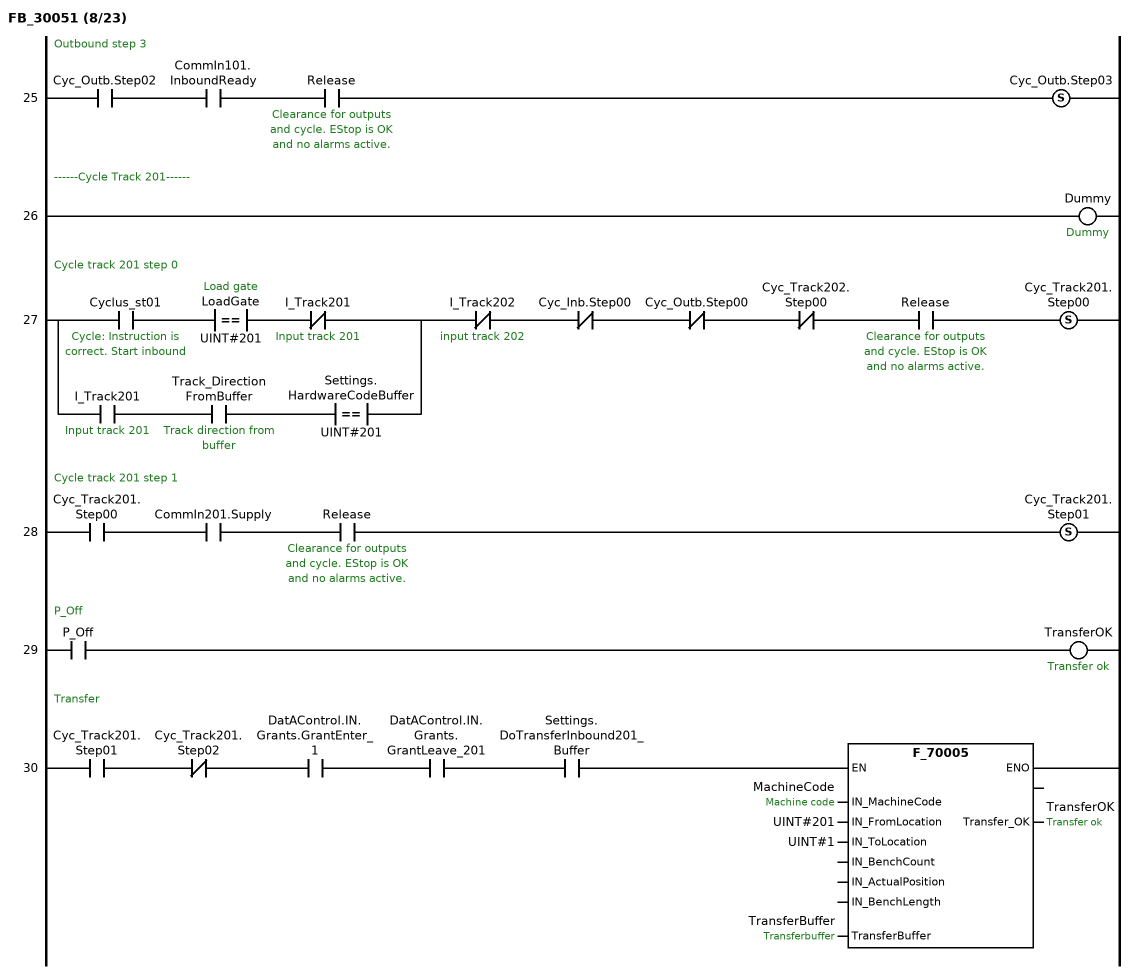
(* Rung 25: Outbound step 3 *)
IF Cyc_Outb.Step02 AND CommIn101.InboundReady AND Release THEN Cyc_Outb.Step03 := TRUE; END_IF;
(* Rung 26: ------Cycle Track 201------ *)
Dummy := TRUE;
(* Rung 27: Cycle track 201 step 0 *)
IF ((Cyclus_st01 AND (LoadGate = UINT#201) AND NOT I_Track201) OR (I_Track201 AND Track_DirectionFromBuffer AND (Settings.HardwareCodeBuffer = UINT#201))) AND NOT I_Track202 AND NOT Cyc_Inb.Step00 AND NOT Cyc_Outb.Step00 AND NOT Cyc_Track202.Step00 AND Release THEN
    Cyc_Track201.Step00 := TRUE;
END_IF;
(* Rung 28: Cycle track 201 step 1 *)
IF Cyc_Track201.Step00 AND CommIn201.Supply AND Release THEN Cyc_Track201.Step01 := TRUE; END_IF;
(* Rung 29: P_Off *)
TransferOK := P_Off;
(* Rung 30: Transfer *)
IF Cyc_Track201.Step01 AND NOT Cyc_Track201.Step02 AND DatAControl.IN.Grants.GrantEnter_1 AND DatAControl.IN.Grants.GrantLeave_201 AND Settings.DoTransferInbound201_Buffer THEN
    F_70005(IN_MachineCode := MachineCode, IN_FromLocation := UINT#201, IN_ToLocation := UINT#1, TransferBuffer := TransferBuffer, Transfer_OK => TransferOK);
END_IF;

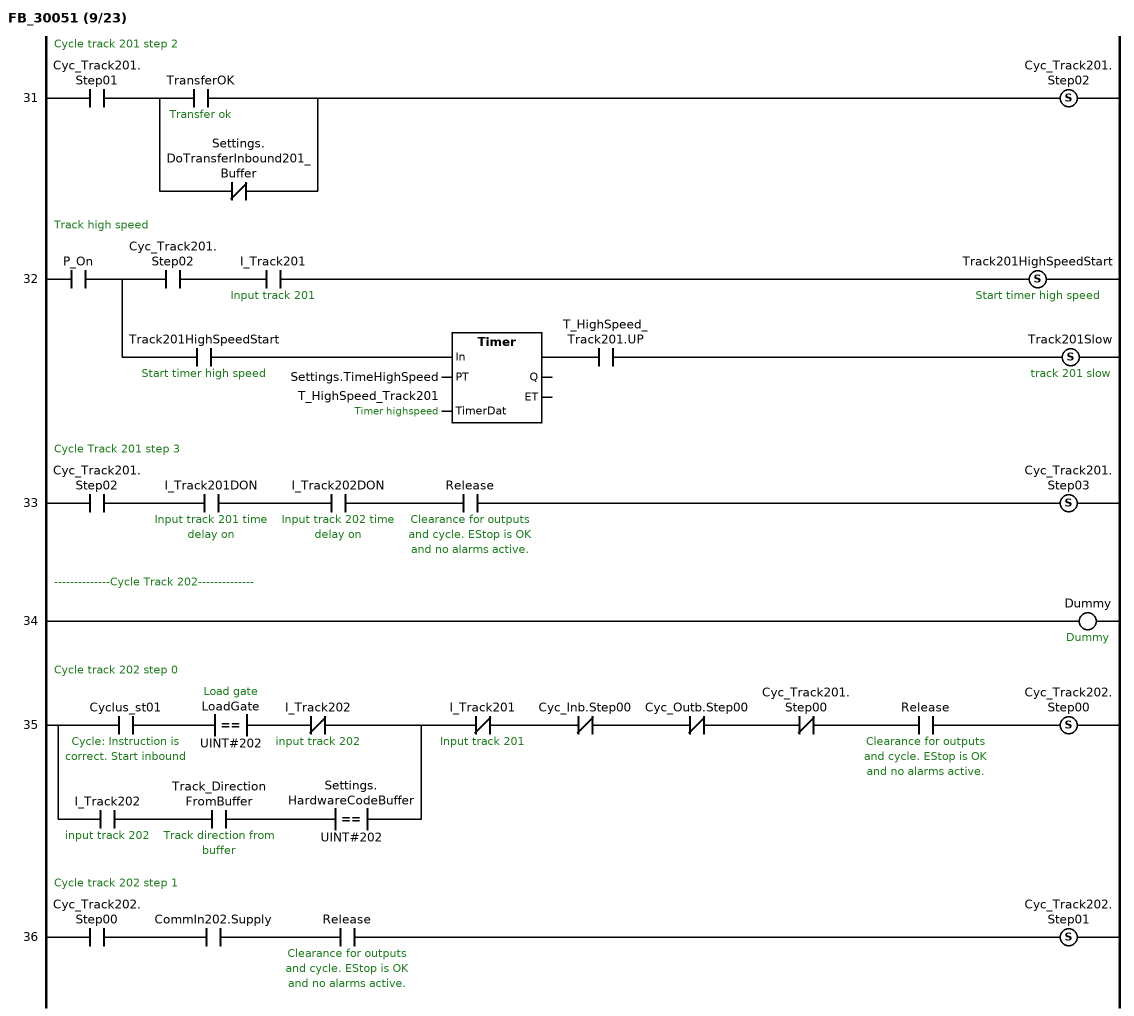
(* Rung 31: Cycle track 201 step 2 *)
IF Cyc_Track201.Step01 AND (TransferOK OR NOT Settings.DoTransferInbound201_Buffer) THEN
    Cyc_Track201.Step02 := TRUE;
END_IF;
(* Rung 32: Track high speed *)
IF P_On AND Cyc_Track201.Step02 AND I_Track201 THEN Track201HighSpeedStart := TRUE; END_IF;
_t2 := Timer(In := P_On AND Track201HighSpeedStart, PT := Settings.TimeHighSpeed, TimerDat := T_HighSpeed_Track201);
IF _t2 AND T_HighSpeed_Track201.UP THEN Track201Slow := TRUE; END_IF;
(* Rung 33: Cycle Track 201 step 3 *)
IF Cyc_Track201.Step02 AND I_Track201DON AND I_Track202DON AND Release THEN
    Cyc_Track201.Step03 := TRUE;
END_IF;
(* Rung 34: --------------Cycle Track 202-------------- *)
Dummy := TRUE;
(* Rung 35: Cycle track 202 step 0 *)
IF ((Cyclus_st01 AND (LoadGate = UINT#202) AND NOT I_Track202) OR (I_Track202 AND Track_DirectionFromBuffer AND (Settings.HardwareCodeBuffer = UINT#202))) AND NOT I_Track201 AND NOT Cyc_Inb.Step00 AND NOT Cyc_Outb.Step00 AND NOT Cyc_Track201.Step00 AND Release THEN
    Cyc_Track202.Step00 := TRUE;
END_IF;
(* Rung 36: Cycle track 202 step 1 *)
IF Cyc_Track202.Step00 AND CommIn202.Supply AND Release THEN Cyc_Track202.Step01 := TRUE; END_IF;

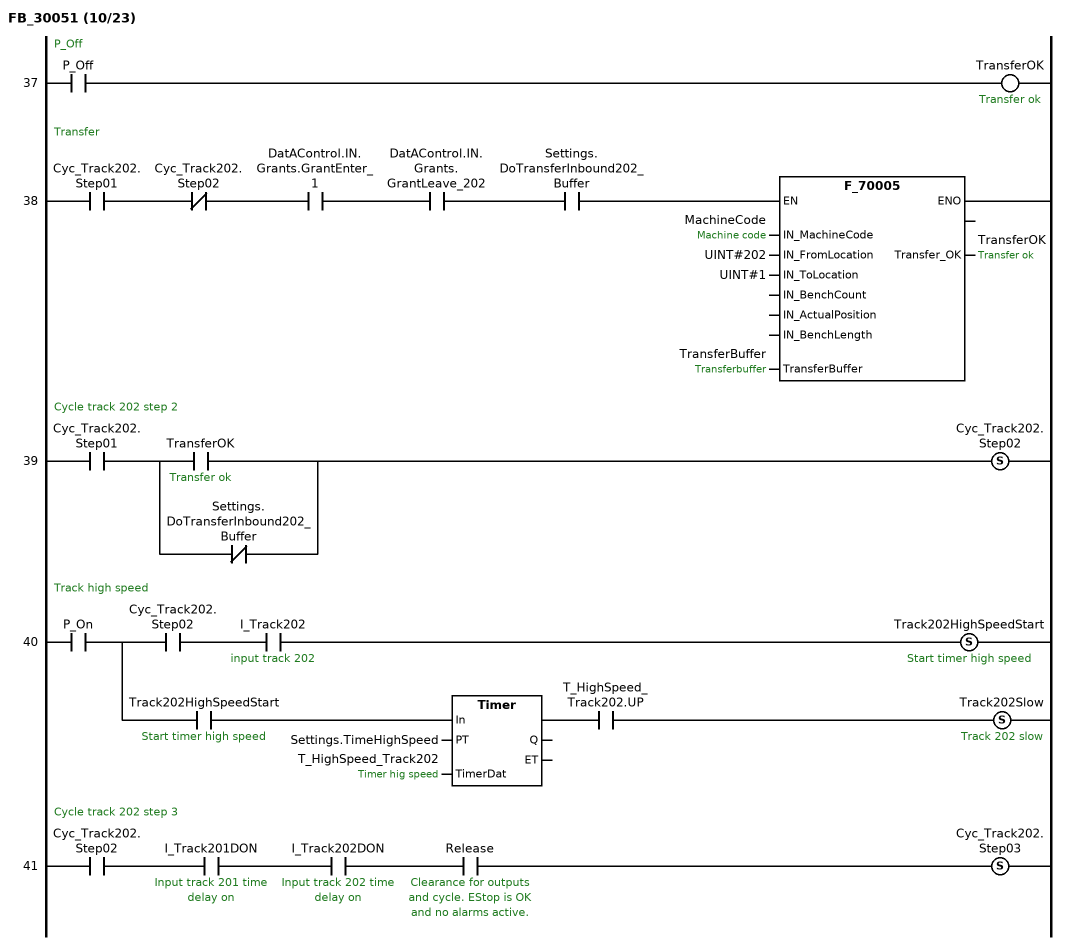
(* Rung 37: P_Off *)
TransferOK := P_Off;
(* Rung 38: Transfer *)
IF Cyc_Track202.Step01 AND NOT Cyc_Track202.Step02 AND DatAControl.IN.Grants.GrantEnter_1 AND DatAControl.IN.Grants.GrantLeave_202 AND Settings.DoTransferInbound202_Buffer THEN
    F_70005(IN_MachineCode := MachineCode, IN_FromLocation := UINT#202, IN_ToLocation := UINT#1, TransferBuffer := TransferBuffer, Transfer_OK => TransferOK);
END_IF;
(* Rung 39: Cycle track 202 step 2 *)
IF Cyc_Track202.Step01 AND (TransferOK OR NOT Settings.DoTransferInbound202_Buffer) THEN
    Cyc_Track202.Step02 := TRUE;
END_IF;
(* Rung 40: Track high speed *)
IF P_On AND Cyc_Track202.Step02 AND I_Track202 THEN Track202HighSpeedStart := TRUE; END_IF;
_t3 := Timer(In := P_On AND Track202HighSpeedStart, PT := Settings.TimeHighSpeed, TimerDat := T_HighSpeed_Track202);
IF _t3 AND T_HighSpeed_Track202.UP THEN Track202Slow := TRUE; END_IF;
(* Rung 41: Cycle track 202 step 3 *)
IF Cyc_Track202.Step02 AND I_Track201DON AND I_Track202DON AND Release THEN
    Cyc_Track202.Step03 := TRUE;
END_IF;

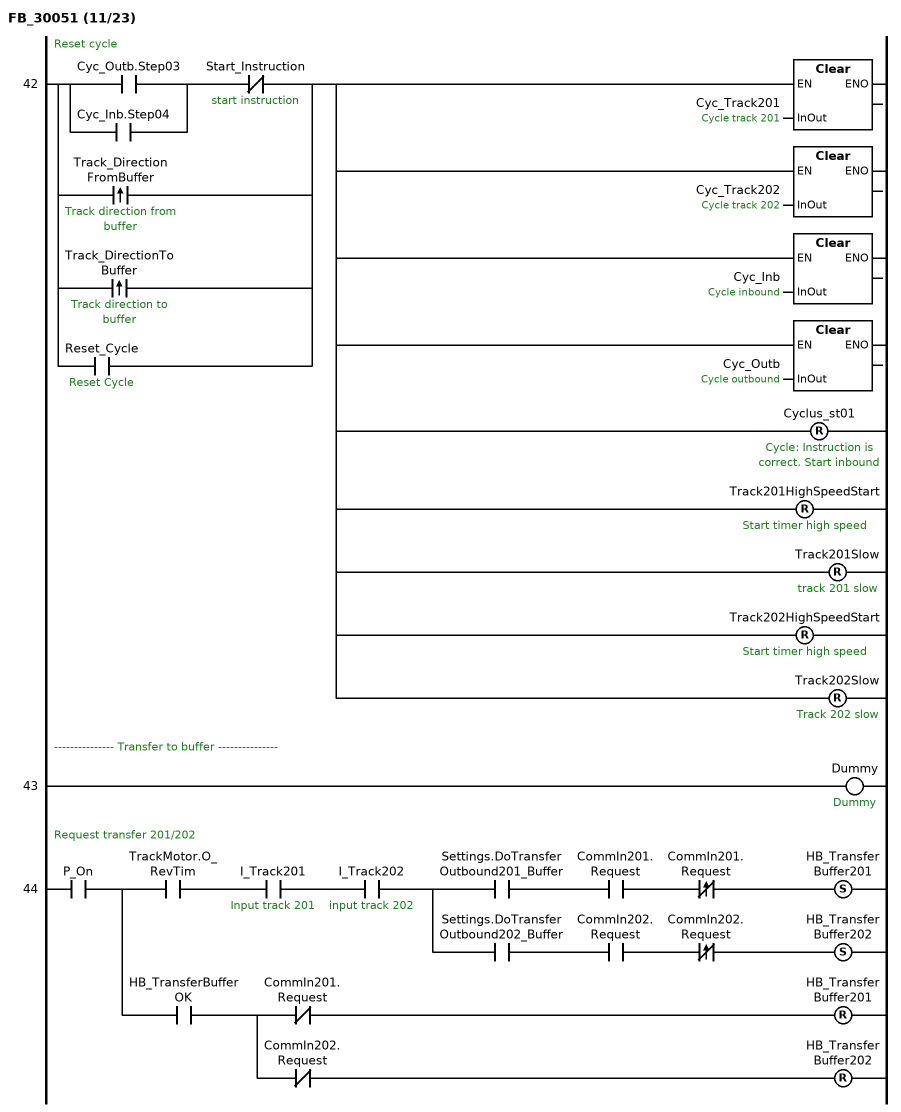
(* Rung 42: Reset cycle *)
_e4(CLK := Track_DirectionFromBuffer);
_e5(CLK := Track_DirectionToBuffer);
_p6 := ((Cyc_Outb.Step03 OR Cyc_Inb.Step04) AND NOT Start_Instruction) OR _e4.Q OR _e5.Q OR Reset_Cycle;
IF _p6 THEN
    Clear(InOut := Cyc_Track201);
    Clear(InOut := Cyc_Track202);
    Clear(InOut := Cyc_Inb);
    Clear(InOut := Cyc_Outb);
    Cyclus_st01 := FALSE;
    Track201HighSpeedStart := FALSE;
    Track201Slow := FALSE;
    Track202HighSpeedStart := FALSE;
    Track202Slow := FALSE;
END_IF;
(* Rung 43: --------------- Transfer to buffer --------------- *)
Dummy := TRUE;
(* Rung 44: Request transfer 201/202 *)
_p7 := P_On AND TrackMotor.O_RevTim AND I_Track201 AND I_Track202;
_e8(CLK := CommIn201.Request);
IF _p7 AND Settings.DoTransferOutbound201_Buffer AND CommIn201.Request AND NOT _e8.Q THEN
    HB_TransferBuffer201 := TRUE;
END_IF;
_e9(CLK := CommIn202.Request);
IF _p7 AND Settings.DoTransferOutbound202_Buffer AND CommIn202.Request AND NOT _e9.Q THEN
    HB_TransferBuffer202 := TRUE;
END_IF;
IF P_On AND HB_TransferBufferOK AND NOT CommIn201.Request THEN HB_TransferBuffer201 := FALSE; END_IF;
IF P_On AND HB_TransferBufferOK AND NOT CommIn202.Request THEN HB_TransferBuffer202 := FALSE; END_IF;

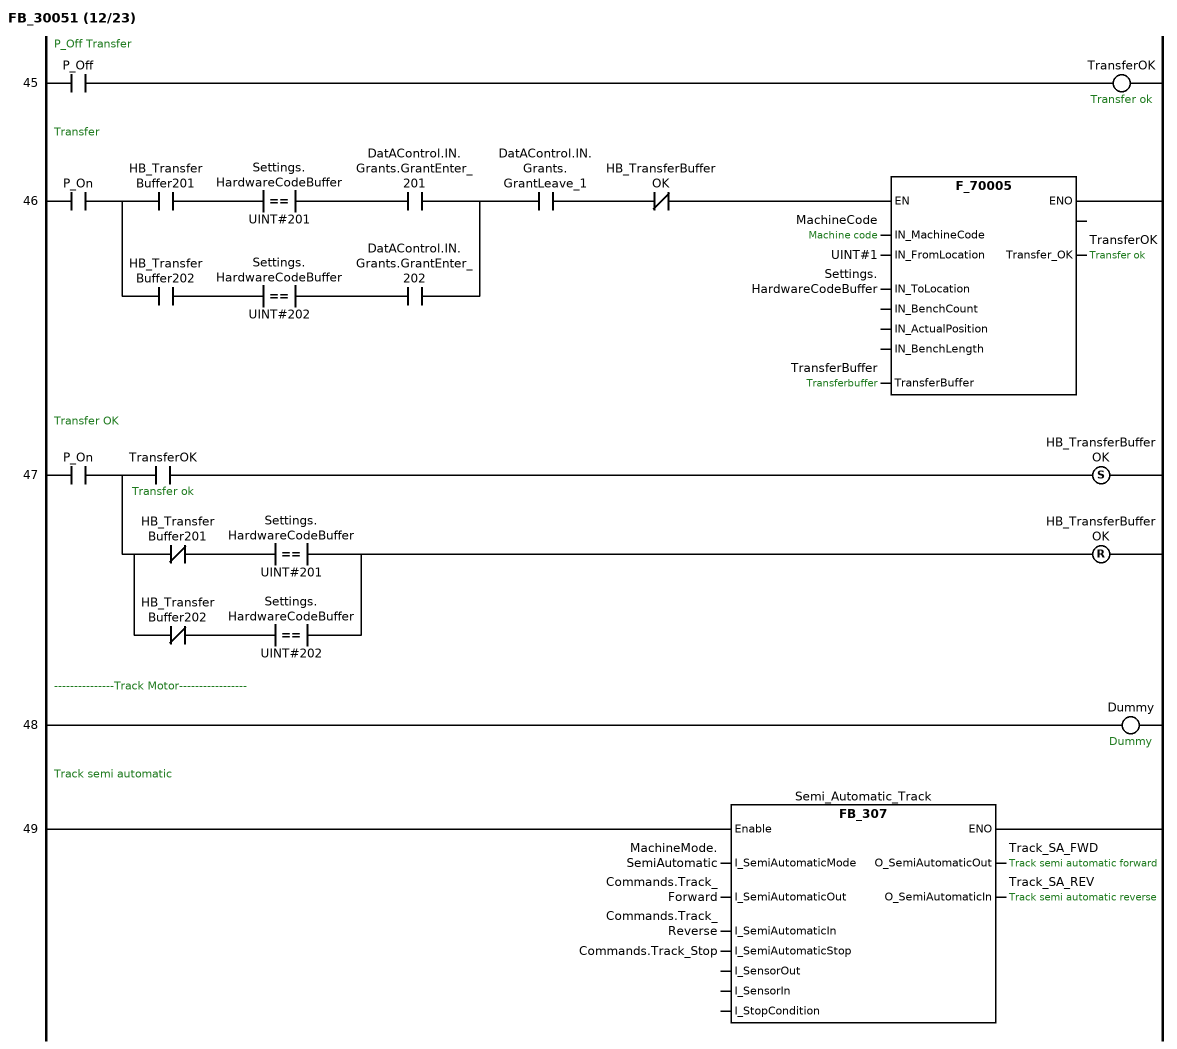
(* Rung 45: P_Off Transfer *)
TransferOK := P_Off;
(* Rung 46: Transfer *)
IF P_On AND ((HB_TransferBuffer201 AND (Settings.HardwareCodeBuffer = UINT#201) AND DatAControl.IN.Grants.GrantEnter_201) OR (HB_TransferBuffer202 AND (Settings.HardwareCodeBuffer = UINT#202) AND DatAControl.IN.Grants.GrantEnter_202)) AND DatAControl.IN.Grants.GrantLeave_1 AND NOT HB_TransferBufferOK THEN
    F_70005(IN_MachineCode := MachineCode, IN_FromLocation := UINT#1, IN_ToLocation := Settings.HardwareCodeBuffer, TransferBuffer := TransferBuffer, Transfer_OK => TransferOK);
END_IF;
(* Rung 47: Transfer OK *)
IF P_On AND TransferOK THEN HB_TransferBufferOK := TRUE; END_IF;
IF P_On AND ((NOT HB_TransferBuffer201 AND (Settings.HardwareCodeBuffer = UINT#201)) OR (NOT HB_TransferBuffer202 AND (Settings.HardwareCodeBuffer = UINT#202))) THEN
    HB_TransferBufferOK := FALSE;
END_IF;
(* Rung 48: ---------------Track Motor----------------- *)
Dummy := TRUE;
(* Rung 49: Track semi automatic *)
Semi_Automatic_Track(Enable := TRUE, I_SemiAutomaticMode := MachineMode.SemiAutomatic, I_SemiAutomaticOut := Commands.Track_Forward, I_SemiAutomaticIn := Commands.Track_Reverse, I_SemiAutomaticStop := Commands.Track_Stop, O_SemiAutomaticOut => Track_SA_FWD, O_SemiAutomaticIn => Track_SA_REV);

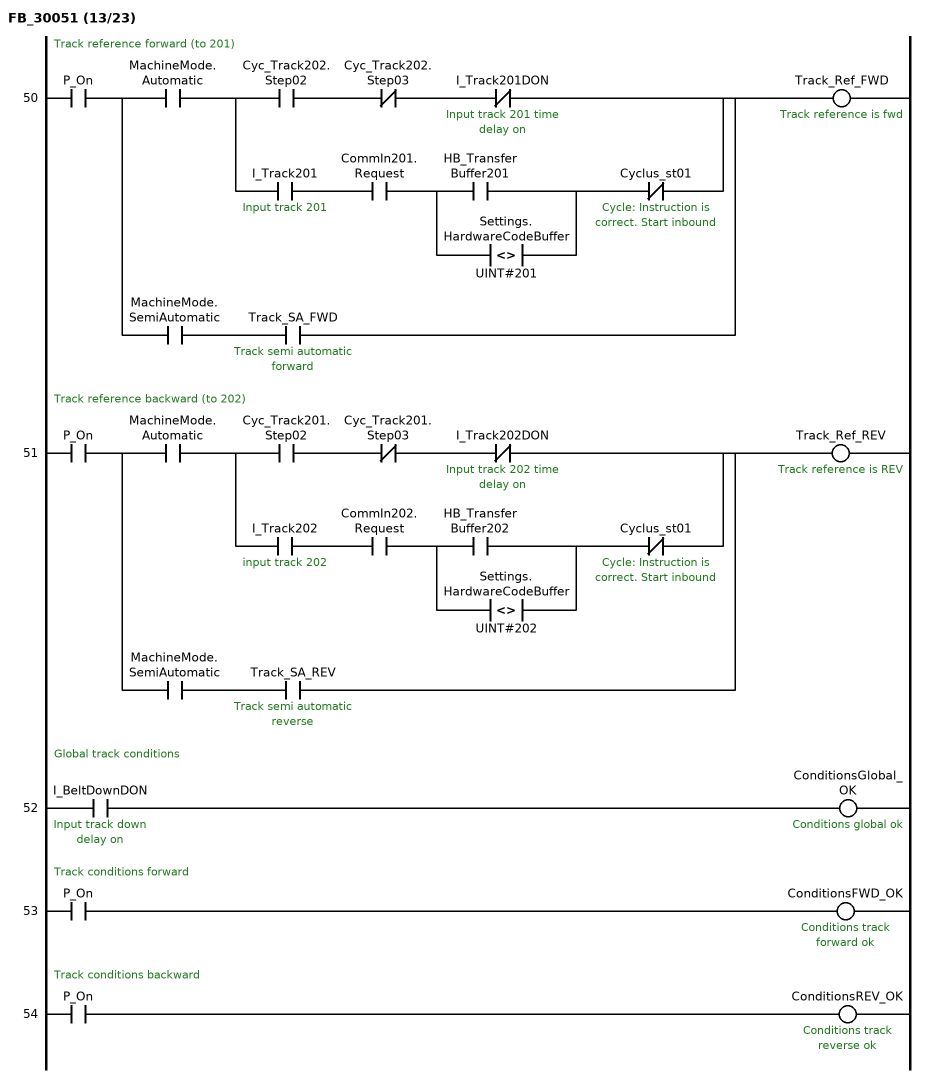
(* Rung 50: Track reference forward (to 201) *)
Track_Ref_FWD := P_On AND ((MachineMode.Automatic AND ((Cyc_Track202.Step02 AND NOT Cyc_Track202.Step03 AND NOT I_Track201DON) OR (I_Track201 AND CommIn201.Request AND (HB_TransferBuffer201 OR (Settings.HardwareCodeBuffer <> UINT#201)) AND NOT Cyclus_st01))) OR (MachineMode.SemiAutomatic AND Track_SA_FWD));
(* Rung 51: Track reference backward (to 202) *)
Track_Ref_REV := P_On AND ((MachineMode.Automatic AND ((Cyc_Track201.Step02 AND NOT Cyc_Track201.Step03 AND NOT I_Track202DON) OR (I_Track202 AND CommIn202.Request AND (HB_TransferBuffer202 OR (Settings.HardwareCodeBuffer <> UINT#202)) AND NOT Cyclus_st01))) OR (MachineMode.SemiAutomatic AND Track_SA_REV));
(* Rung 52: Global track conditions *)
ConditionsGlobal_OK := I_BeltDownDON;
(* Rung 53: Track conditions forward *)
ConditionsFWD_OK := P_On;
(* Rung 54: Track conditions backward *)
ConditionsREV_OK := P_On;

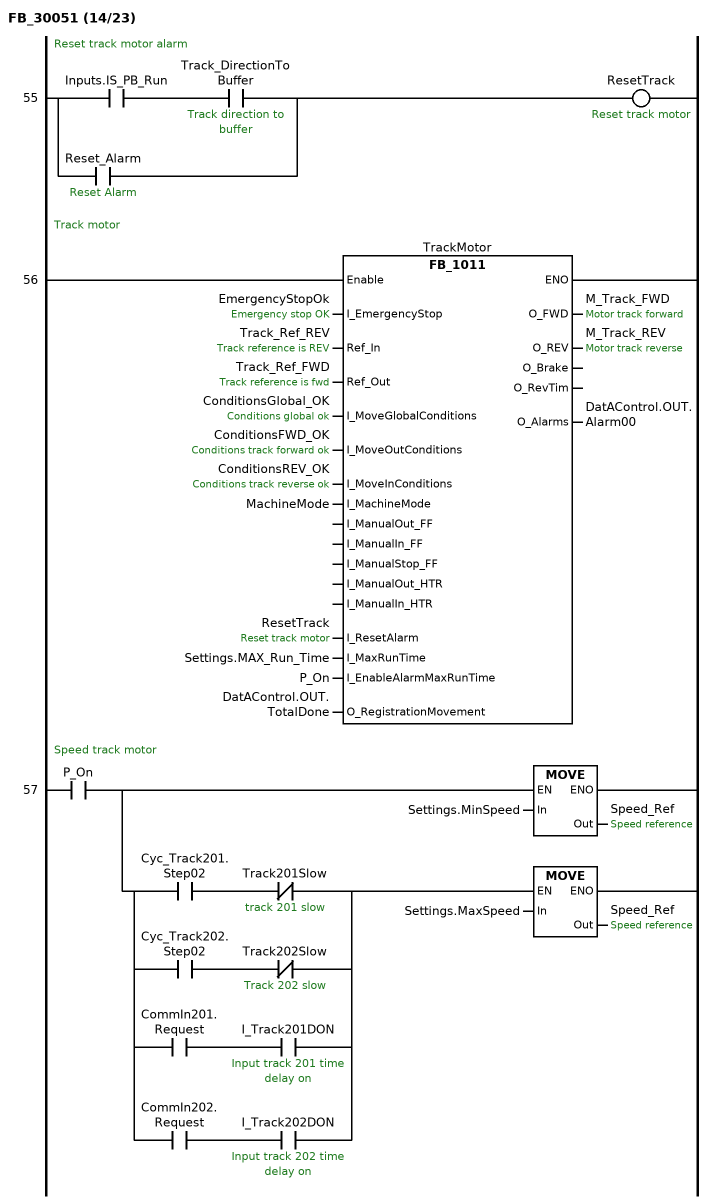
(* Rung 55: Reset track motor alarm *)
ResetTrack := (Inputs.IS_PB_Run AND Track_DirectionToBuffer) OR Reset_Alarm;
(* Rung 56: Track motor *)
TrackMotor(Enable := TRUE, I_EmergencyStop := EmergencyStopOk, Ref_In := Track_Ref_REV, Ref_Out := Track_Ref_FWD, I_MoveGlobalConditions := ConditionsGlobal_OK, I_MoveOutConditions := ConditionsFWD_OK, I_MoveInConditions := ConditionsREV_OK, I_MachineMode := MachineMode, I_ResetAlarm := ResetTrack, I_MaxRunTime := Settings.MAX_Run_Time, I_EnableAlarmMaxRunTime := P_On, O_RegistrationMovement := DatAControl.OUT.TotalDone, O_FWD => M_Track_FWD, O_REV => M_Track_REV, O_Alarms => DatAControl.OUT.Alarm00);
(* Rung 57: Speed track motor *)
IF P_On THEN Speed_Ref := Settings.MinSpeed; END_IF;
IF P_On AND ((Cyc_Track201.Step02 AND NOT Track201Slow) OR (Cyc_Track202.Step02 AND NOT Track202Slow) OR (CommIn201.Request AND I_Track201DON) OR (CommIn202.Request AND I_Track202DON)) THEN
    Speed_Ref := Settings.MaxSpeed;
END_IF;

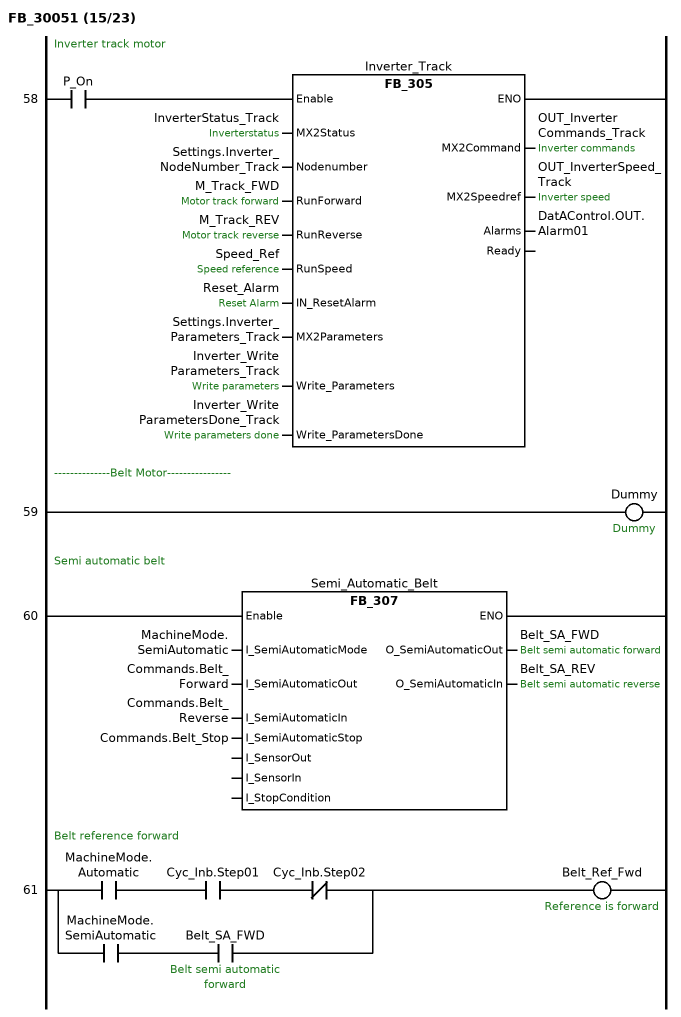
(* Rung 58: Inverter track motor *)
Inverter_Track(Enable := P_On, MX2Status := InverterStatus_Track, Nodenumber := Settings.Inverter_NodeNumber_Track, RunForward := M_Track_FWD, RunReverse := M_Track_REV, RunSpeed := Speed_Ref, IN_ResetAlarm := Reset_Alarm, MX2Parameters := Settings.Inverter_Parameters_Track, Write_Parameters := Inverter_WriteParameters_Track, Write_ParametersDone := Inverter_WriteParametersDone_Track, MX2Command => OUT_InverterCommands_Track, MX2Speedref => OUT_InverterSpeed_Track, Alarms => DatAControl.OUT.Alarm01);
(* Rung 59: --------------Belt Motor---------------- *)
Dummy := TRUE;
(* Rung 60: Semi automatic belt *)
Semi_Automatic_Belt(Enable := TRUE, I_SemiAutomaticMode := MachineMode.SemiAutomatic, I_SemiAutomaticOut := Commands.Belt_Forward, I_SemiAutomaticIn := Commands.Belt_Reverse, I_SemiAutomaticStop := Commands.Belt_Stop, O_SemiAutomaticOut => Belt_SA_FWD, O_SemiAutomaticIn => Belt_SA_REV);
(* Rung 61: Belt reference forward *)
Belt_Ref_Fwd := (MachineMode.Automatic AND Cyc_Inb.Step01 AND NOT Cyc_Inb.Step02) OR (MachineMode.SemiAutomatic AND Belt_SA_FWD);

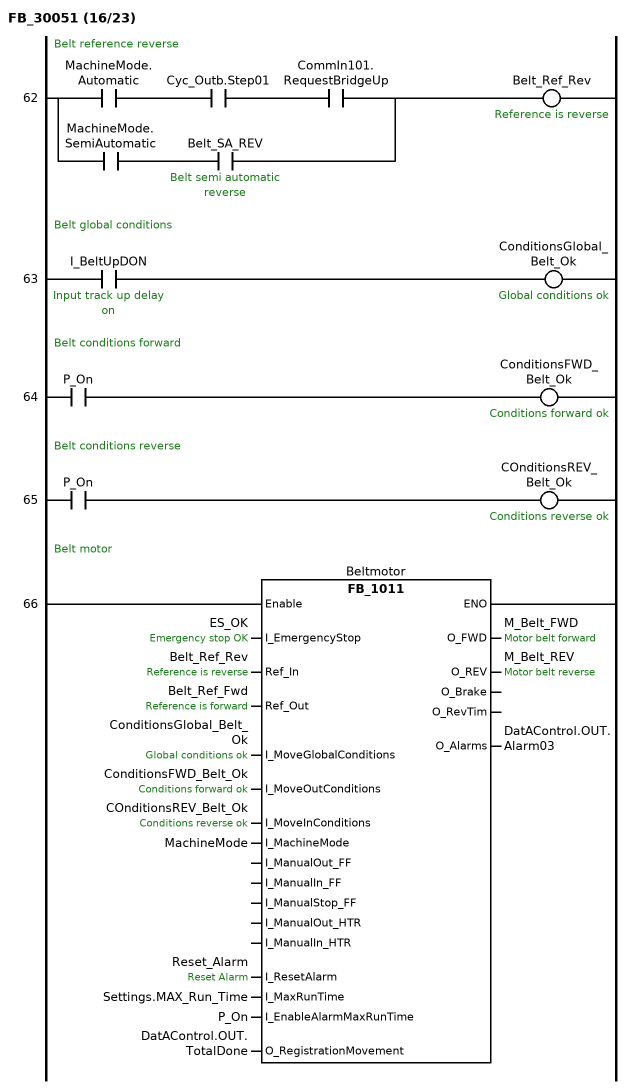
(* Rung 62: Belt reference reverse *)
Belt_Ref_Rev := (MachineMode.Automatic AND Cyc_Outb.Step01 AND CommIn101.RequestBridgeUp) OR (MachineMode.SemiAutomatic AND Belt_SA_REV);
(* Rung 63: Belt global conditions *)
ConditionsGlobal_Belt_Ok := I_BeltUpDON;
(* Rung 64: Belt conditions forward *)
ConditionsFWD_Belt_Ok := P_On;
(* Rung 65: Belt conditions reverse *)
COnditionsREV_Belt_Ok := P_On;
(* Rung 66: Belt motor *)
Beltmotor(Enable := TRUE, I_EmergencyStop := ES_OK, Ref_In := Belt_Ref_Rev, Ref_Out := Belt_Ref_Fwd, I_MoveGlobalConditions := ConditionsGlobal_Belt_Ok, I_MoveOutConditions := ConditionsFWD_Belt_Ok, I_MoveInConditions := COnditionsREV_Belt_Ok, I_MachineMode := MachineMode, I_ResetAlarm := Reset_Alarm, I_MaxRunTime := Settings.MAX_Run_Time, I_EnableAlarmMaxRunTime := P_On, O_RegistrationMovement := DatAControl.OUT.TotalDone, O_FWD => M_Belt_FWD, O_REV => M_Belt_REV, O_Alarms => DatAControl.OUT.Alarm03);

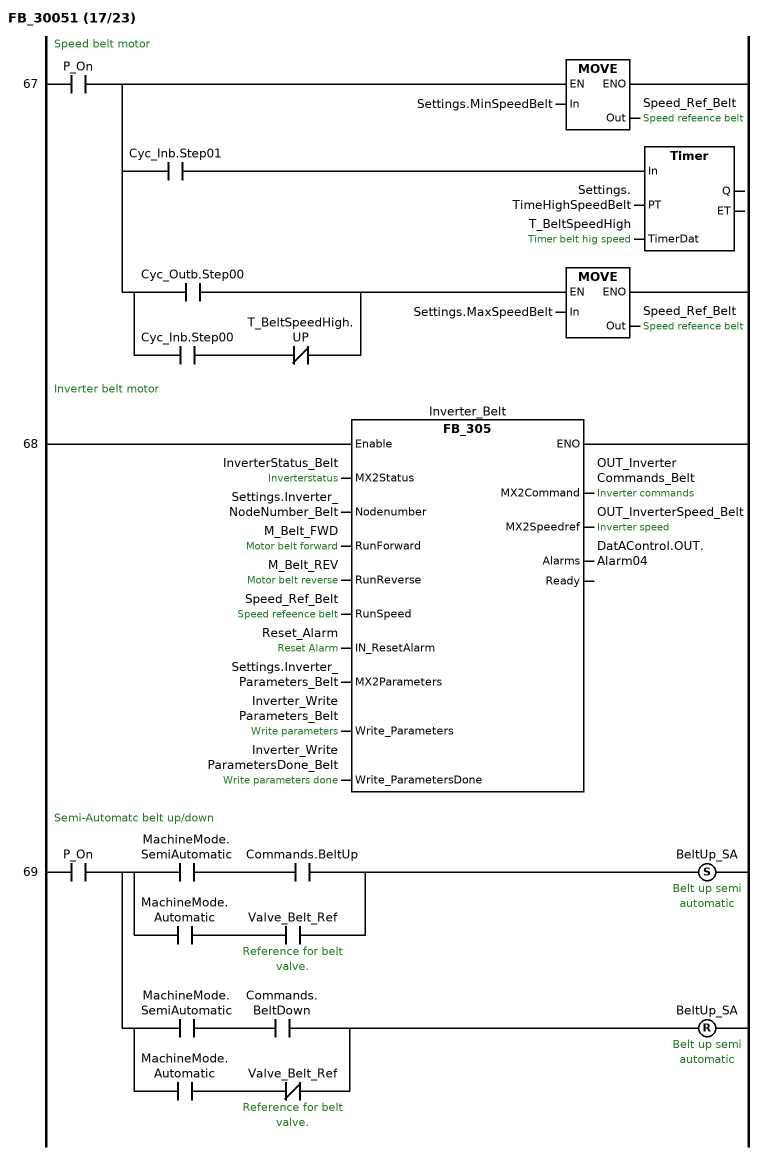
(* Rung 67: Speed belt motor *)
IF P_On THEN Speed_Ref_Belt := Settings.MinSpeedBelt; END_IF;
_t10 := Timer(In := P_On AND Cyc_Inb.Step01, PT := Settings.TimeHighSpeedBelt, TimerDat := T_BeltSpeedHigh);
IF P_On AND (Cyc_Outb.Step00 OR (Cyc_Inb.Step00 AND NOT T_BeltSpeedHigh.UP)) THEN
    Speed_Ref_Belt := Settings.MaxSpeedBelt;
END_IF;
(* Rung 68: Inverter belt motor *)
Inverter_Belt(Enable := TRUE, MX2Status := InverterStatus_Belt, Nodenumber := Settings.Inverter_NodeNumber_Belt, RunForward := M_Belt_FWD, RunReverse := M_Belt_REV, RunSpeed := Speed_Ref_Belt, IN_ResetAlarm := Reset_Alarm, MX2Parameters := Settings.Inverter_Parameters_Belt, Write_Parameters := Inverter_WriteParameters_Belt, Write_ParametersDone := Inverter_WriteParametersDone_Belt, MX2Command => OUT_InverterCommands_Belt, MX2Speedref => OUT_InverterSpeed_Belt, Alarms => DatAControl.OUT.Alarm04);
(* Rung 69: Semi-Automatc belt up/down *)
IF P_On AND ((MachineMode.SemiAutomatic AND Commands.BeltUp) OR (MachineMode.Automatic AND Valve_Belt_Ref)) THEN
    BeltUp_SA := TRUE;
END_IF;
IF P_On AND ((MachineMode.SemiAutomatic AND Commands.BeltDown) OR (MachineMode.Automatic AND NOT Valve_Belt_Ref)) THEN
    BeltUp_SA := FALSE;
END_IF;

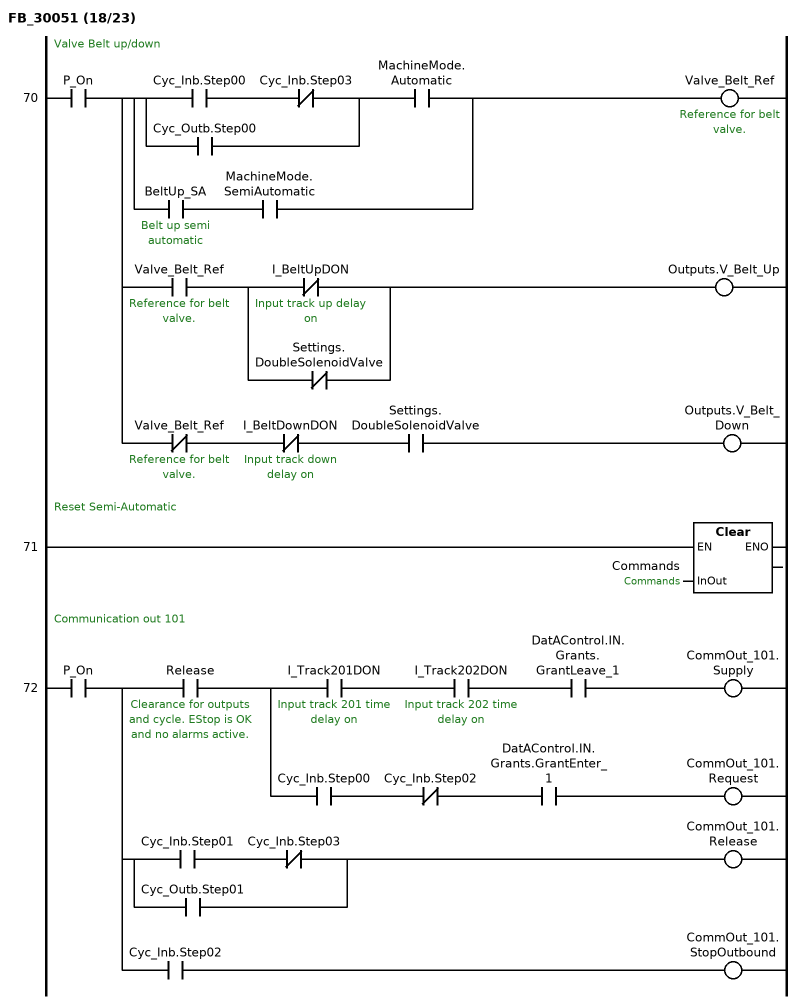
(* Rung 70: Valve Belt up/down *)
Valve_Belt_Ref := P_On AND ((((Cyc_Inb.Step00 AND NOT Cyc_Inb.Step03) OR Cyc_Outb.Step00) AND MachineMode.Automatic) OR (BeltUp_SA AND MachineMode.SemiAutomatic));
Outputs.V_Belt_Up := P_On AND Valve_Belt_Ref AND (NOT I_BeltUpDON OR NOT Settings.DoubleSolenoidValve);
Outputs.V_Belt_Down := P_On AND NOT Valve_Belt_Ref AND NOT I_BeltDownDON AND Settings.DoubleSolenoidValve;
(* Rung 71: Reset Semi-Automatic *)
Clear(InOut := Commands);
(* Rung 72: Communication out 101 *)
CommOut_101.Supply := P_On AND Release AND I_Track201DON AND I_Track202DON AND DatAControl.IN.Grants.GrantLeave_1;
CommOut_101.Request := P_On AND Release AND Cyc_Inb.Step00 AND NOT Cyc_Inb.Step02 AND DatAControl.IN.Grants.GrantEnter_1;
CommOut_101.Release := P_On AND ((Cyc_Inb.Step01 AND NOT Cyc_Inb.Step03) OR Cyc_Outb.Step01);
CommOut_101.StopOutbound := P_On AND Cyc_Inb.Step02;

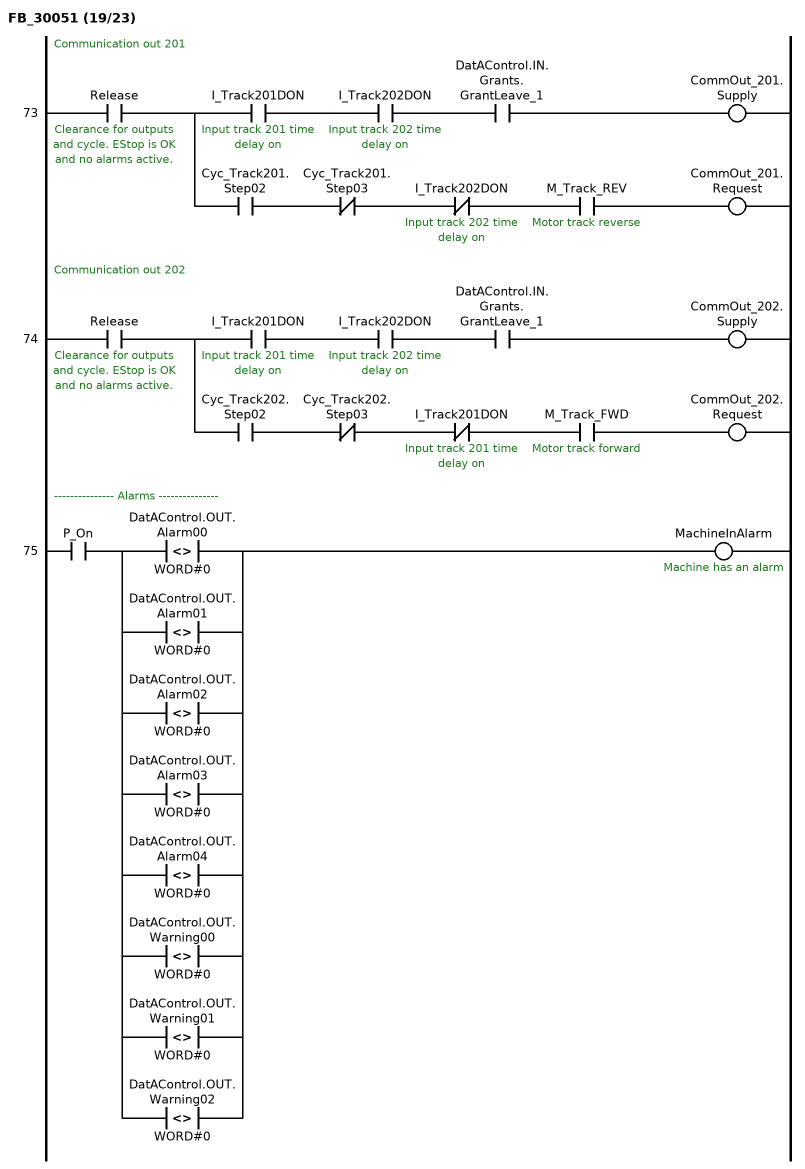
(* Rung 73: Communication out 201 *)
CommOut_201.Supply := Release AND I_Track201DON AND I_Track202DON AND DatAControl.IN.Grants.GrantLeave_1;
CommOut_201.Request := Release AND Cyc_Track201.Step02 AND NOT Cyc_Track201.Step03 AND NOT I_Track202DON AND M_Track_REV;
(* Rung 74: Communication out 202 *)
CommOut_202.Supply := Release AND I_Track201DON AND I_Track202DON AND DatAControl.IN.Grants.GrantLeave_1;
CommOut_202.Request := Release AND Cyc_Track202.Step02 AND NOT Cyc_Track202.Step03 AND NOT I_Track201DON AND M_Track_FWD;
(* Rung 75: --------------- Alarms --------------- *)
MachineInAlarm := P_On AND ((DatAControl.OUT.Alarm00 <> WORD#0) OR (DatAControl.OUT.Alarm01 <> WORD#0) OR (DatAControl.OUT.Alarm02 <> WORD#0) OR (DatAControl.OUT.Alarm03 <> WORD#0) OR (DatAControl.OUT.Alarm04 <> WORD#0) OR (DatAControl.OUT.Warning00 <> WORD#0) OR (DatAControl.OUT.Warning01 <> WORD#0) OR (DatAControl.OUT.Warning02 <> WORD#0));

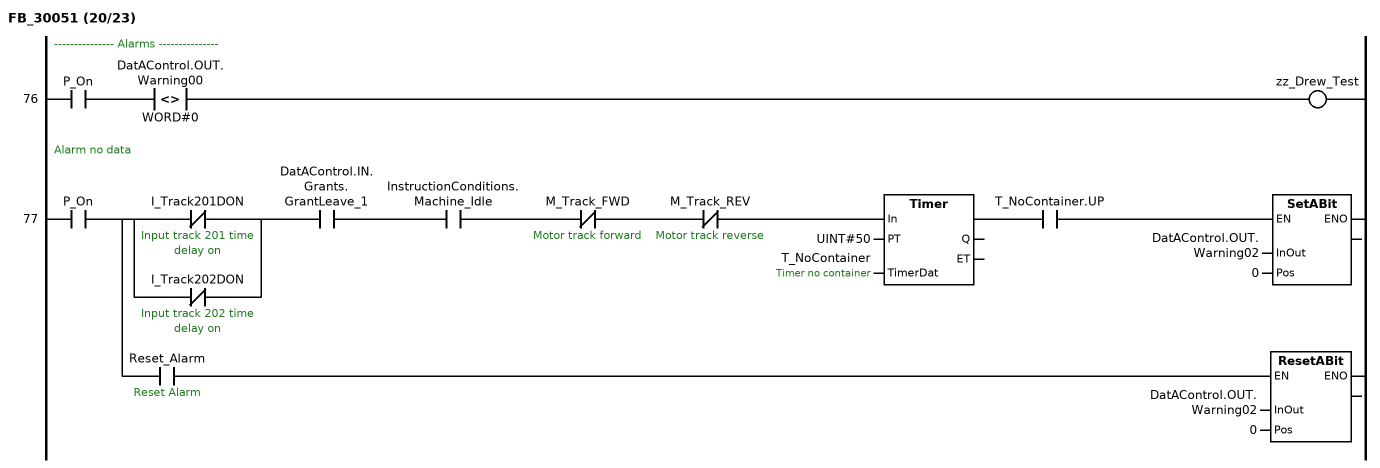
(* Rung 76: --------------- Alarms --------------- *)
zz_Drew_Test := P_On AND (DatAControl.OUT.Warning00 <> WORD#0);
(* Rung 77: Alarm no data *)
_t11 := Timer(In := P_On AND (NOT I_Track201DON OR NOT I_Track202DON) AND DatAControl.IN.Grants.GrantLeave_1 AND InstructionConditions.Machine_Idle AND NOT M_Track_FWD AND NOT M_Track_REV, PT := UINT#50, TimerDat := T_NoContainer);
IF _t11 AND T_NoContainer.UP THEN SetABit(InOut := DatAControl.OUT.Warning02, Pos := 0); END_IF;
IF P_On AND Reset_Alarm THEN ResetABit(InOut := DatAControl.OUT.Warning02, Pos := 0); END_IF;

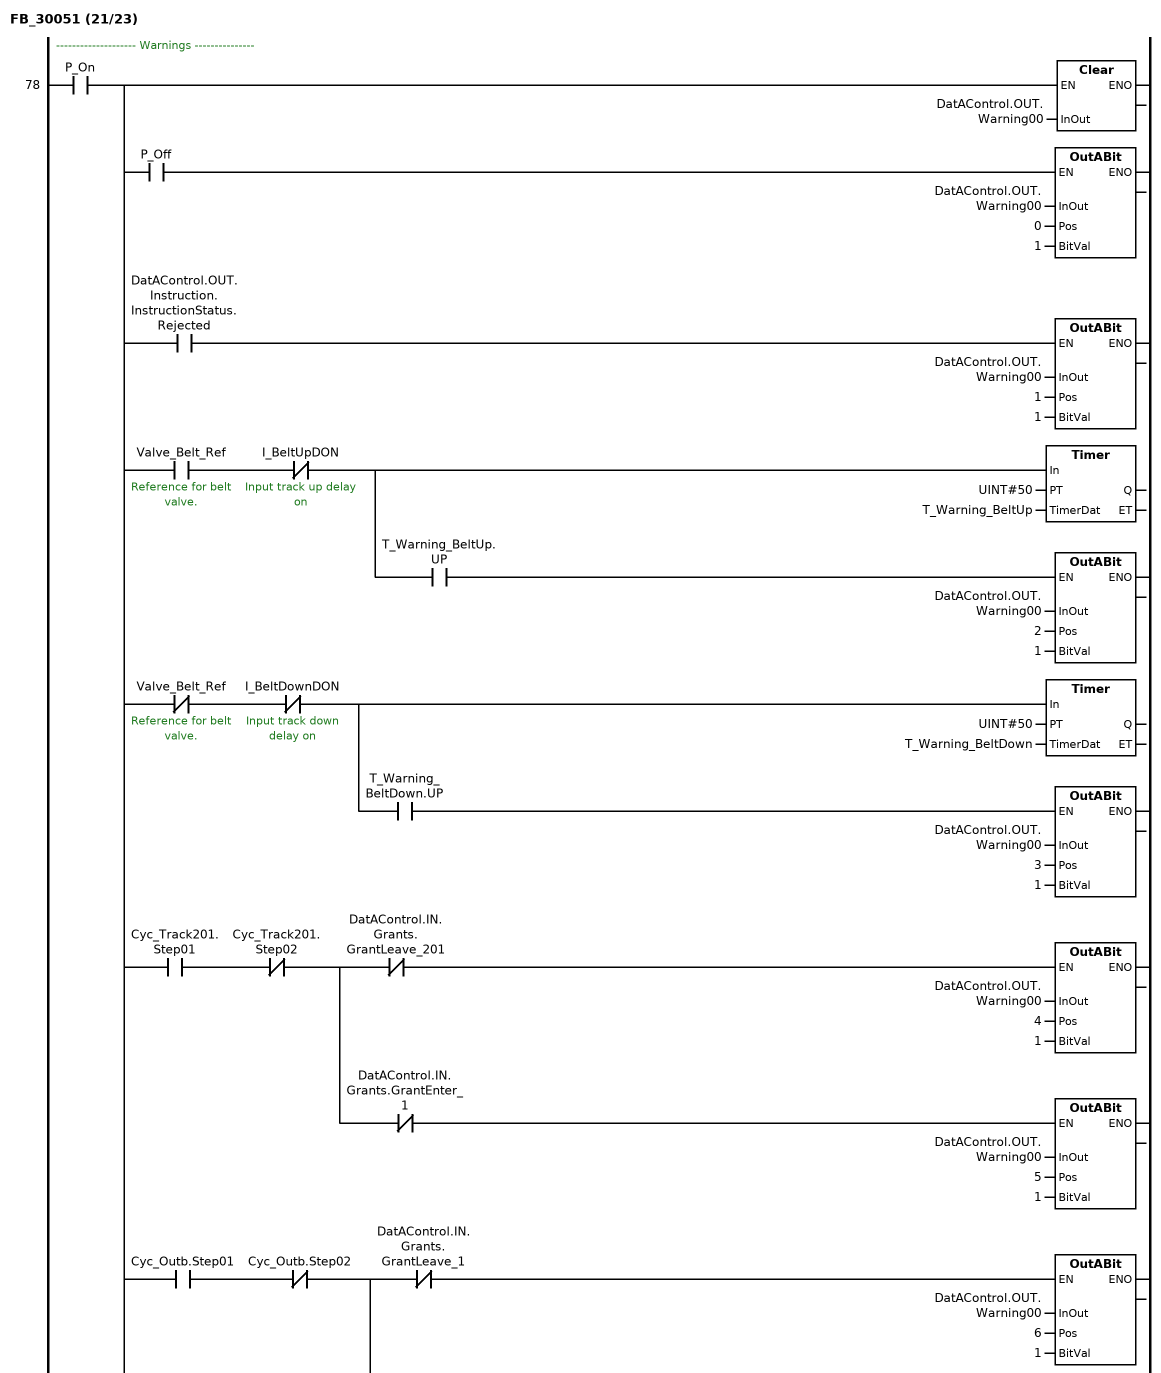

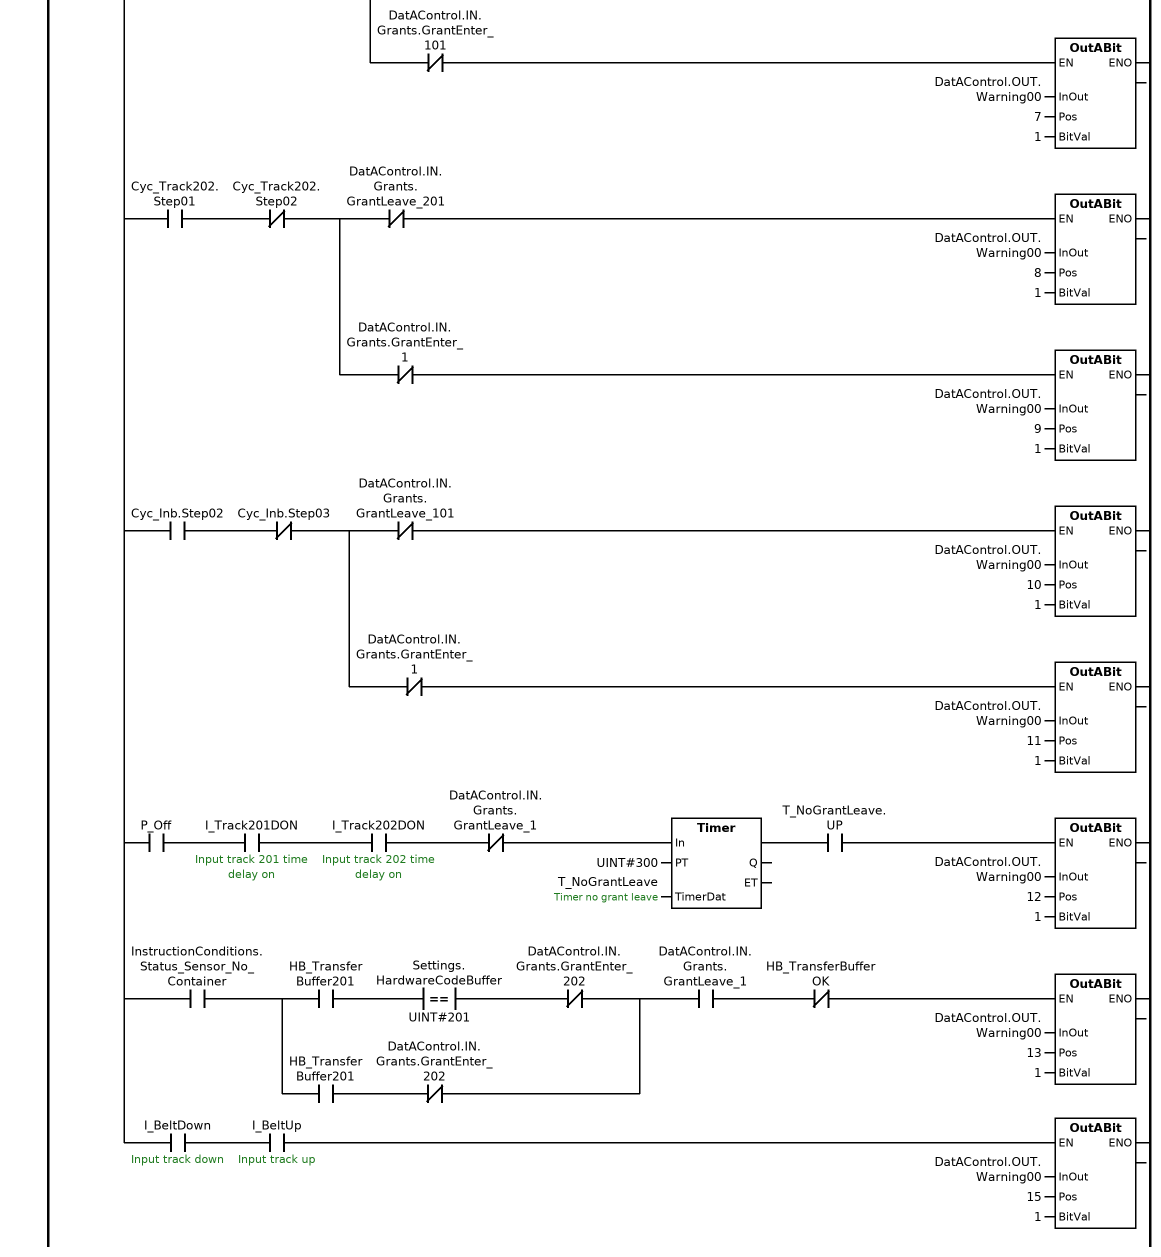
(* Rung 78: -------------------- Warnings --------------- *)
IF P_On THEN Clear(InOut := DatAControl.OUT.Warning00); END_IF;
IF P_On AND P_Off THEN OutABit(InOut := DatAControl.OUT.Warning00, Pos := 0, BitVal := 1); END_IF;
IF P_On AND DatAControl.OUT.Instruction.InstructionStatus.Rejected THEN
    OutABit(InOut := DatAControl.OUT.Warning00, Pos := 1, BitVal := 1);
END_IF;
_t12 := Timer(In := P_On AND Valve_Belt_Ref AND NOT I_BeltUpDON, PT := UINT#50, TimerDat := T_Warning_BeltUp);
IF P_On AND Valve_Belt_Ref AND NOT I_BeltUpDON AND T_Warning_BeltUp.UP THEN
    OutABit(InOut := DatAControl.OUT.Warning00, Pos := 2, BitVal := 1);
END_IF;
_p13 := P_On AND NOT Valve_Belt_Ref AND NOT I_BeltDownDON;
_t14 := Timer(In := _p13, PT := UINT#50, TimerDat := T_Warning_BeltDown);
IF _p13 AND T_Warning_BeltDown.UP THEN
    OutABit(InOut := DatAControl.OUT.Warning00, Pos := 3, BitVal := 1);
END_IF;
_p15 := P_On AND Cyc_Track201.Step01 AND NOT Cyc_Track201.Step02;
IF _p15 AND NOT DatAControl.IN.Grants.GrantLeave_201 THEN
    OutABit(InOut := DatAControl.OUT.Warning00, Pos := 4, BitVal := 1);
END_IF;
IF _p15 AND NOT DatAControl.IN.Grants.GrantEnter_1 THEN
    OutABit(InOut := DatAControl.OUT.Warning00, Pos := 5, BitVal := 1);
END_IF;
IF P_On AND Cyc_Outb.Step01 AND NOT Cyc_Outb.Step02 AND NOT DatAControl.IN.Grants.GrantLeave_1 THEN
    OutABit(InOut := DatAControl.OUT.Warning00, Pos := 6, BitVal := 1);
END_IF;
IF P_On AND Cyc_Outb.Step01 AND NOT Cyc_Outb.Step02 AND NOT DatAControl.IN.Grants.GrantEnter_101 THEN
    OutABit(InOut := DatAControl.OUT.Warning00, Pos := 7, BitVal := 1);
END_IF;
_p16 := P_On AND Cyc_Track202.Step01 AND NOT Cyc_Track202.Step02;
IF _p16 AND NOT DatAControl.IN.Grants.GrantLeave_201 THEN
    OutABit(InOut := DatAControl.OUT.Warning00, Pos := 8, BitVal := 1);
END_IF;
IF _p16 AND NOT DatAControl.IN.Grants.GrantEnter_1 THEN
    OutABit(InOut := DatAControl.OUT.Warning00, Pos := 9, BitVal := 1);
END_IF;
IF P_On AND Cyc_Inb.Step02 AND NOT Cyc_Inb.Step03 AND NOT DatAControl.IN.Grants.GrantLeave_101 THEN
    OutABit(InOut := DatAControl.OUT.Warning00, Pos := 10, BitVal := 1);
END_IF;
IF P_On AND Cyc_Inb.Step02 AND NOT Cyc_Inb.Step03 AND NOT DatAControl.IN.Grants.GrantEnter_1 THEN
    OutABit(InOut := DatAControl.OUT.Warning00, Pos := 11, BitVal := 1);
END_IF;
_t17 := Timer(In := P_On AND P_Off AND I_Track201DON AND I_Track202DON AND NOT DatAControl.IN.Grants.GrantLeave_1, PT := UINT#300, TimerDat := T_NoGrantLeave);
IF _t17 AND T_NoGrantLeave.UP THEN
    OutABit(InOut := DatAControl.OUT.Warning00, Pos := 12, BitVal := 1);
END_IF;
IF P_On AND InstructionConditions.Status_Sensor_No_Container AND ((HB_TransferBuffer201 AND (Settings.HardwareCodeBuffer = UINT#201) AND NOT DatAControl.IN.Grants.GrantEnter_202) OR (HB_TransferBuffer201 AND NOT DatAControl.IN.Grants.GrantEnter_202)) AND DatAControl.IN.Grants.GrantLeave_1 AND NOT HB_TransferBufferOK THEN
    OutABit(InOut := DatAControl.OUT.Warning00, Pos := 13, BitVal := 1);
END_IF;
IF P_On AND I_BeltDown AND I_BeltUp THEN
    OutABit(InOut := DatAControl.OUT.Warning00, Pos := 15, BitVal := 1);
END_IF;

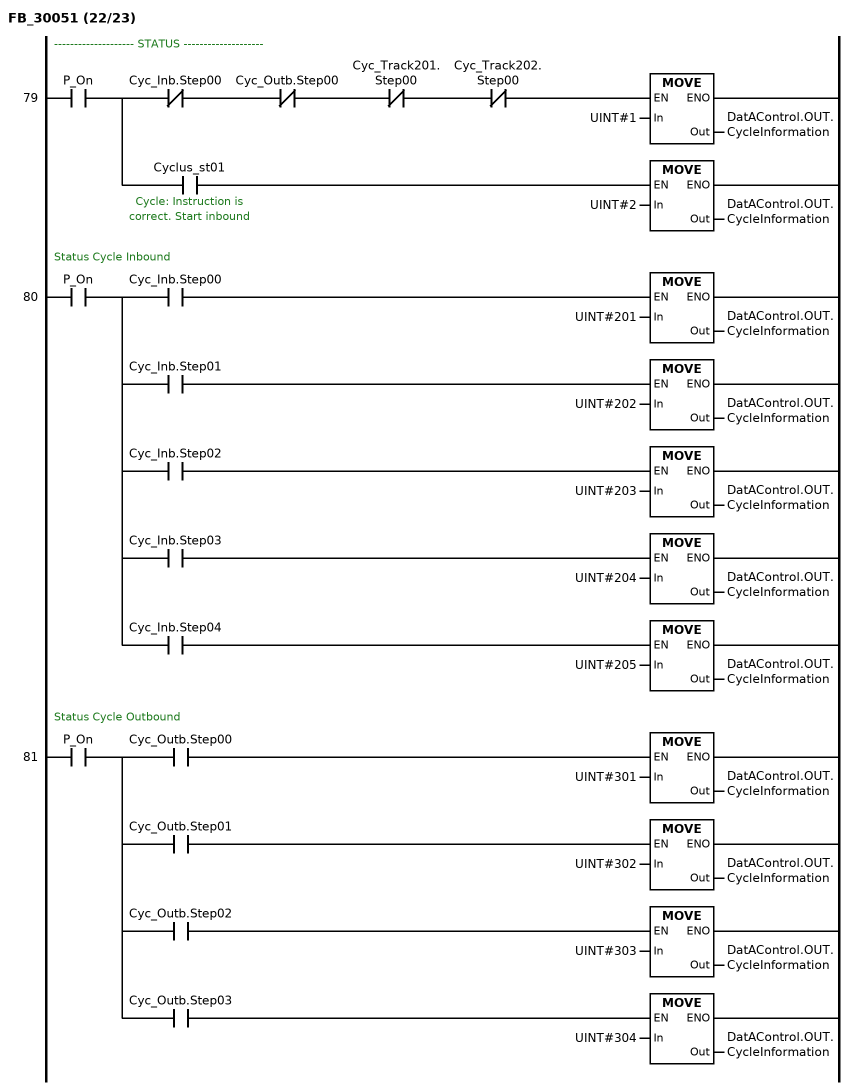
(* Rung 79: -------------------- STATUS -------------------- *)
IF P_On AND NOT Cyc_Inb.Step00 AND NOT Cyc_Outb.Step00 AND NOT Cyc_Track201.Step00 AND NOT Cyc_Track202.Step00 THEN
    DatAControl.OUT.CycleInformation := UINT#1;
END_IF;
IF P_On AND Cyclus_st01 THEN DatAControl.OUT.CycleInformation := UINT#2; END_IF;
(* Rung 80: Status Cycle Inbound *)
IF P_On AND Cyc_Inb.Step00 THEN DatAControl.OUT.CycleInformation := UINT#201; END_IF;
IF P_On AND Cyc_Inb.Step01 THEN DatAControl.OUT.CycleInformation := UINT#202; END_IF;
IF P_On AND Cyc_Inb.Step02 THEN DatAControl.OUT.CycleInformation := UINT#203; END_IF;
IF P_On AND Cyc_Inb.Step03 THEN DatAControl.OUT.CycleInformation := UINT#204; END_IF;
IF P_On AND Cyc_Inb.Step04 THEN DatAControl.OUT.CycleInformation := UINT#205; END_IF;
(* Rung 81: Status Cycle Outbound *)
IF P_On AND Cyc_Outb.Step00 THEN DatAControl.OUT.CycleInformation := UINT#301; END_IF;
IF P_On AND Cyc_Outb.Step01 THEN DatAControl.OUT.CycleInformation := UINT#302; END_IF;
IF P_On AND Cyc_Outb.Step02 THEN DatAControl.OUT.CycleInformation := UINT#303; END_IF;
IF P_On AND Cyc_Outb.Step03 THEN DatAControl.OUT.CycleInformation := UINT#304; END_IF;

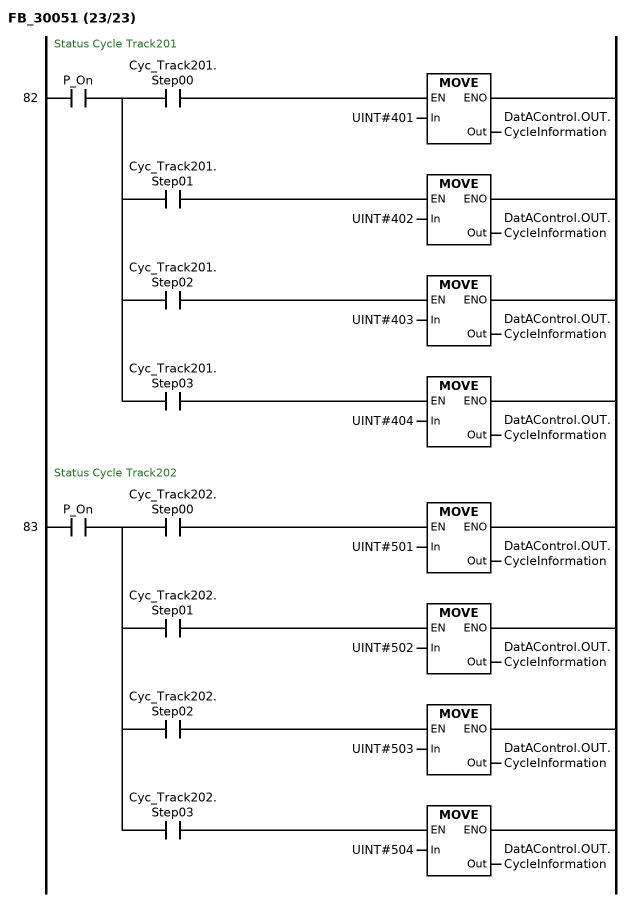
(* Rung 82: Status Cycle Track201 *)
IF P_On AND Cyc_Track201.Step00 THEN DatAControl.OUT.CycleInformation := UINT#401; END_IF;
IF P_On AND Cyc_Track201.Step01 THEN DatAControl.OUT.CycleInformation := UINT#402; END_IF;
IF P_On AND Cyc_Track201.Step02 THEN DatAControl.OUT.CycleInformation := UINT#403; END_IF;
IF P_On AND Cyc_Track201.Step03 THEN DatAControl.OUT.CycleInformation := UINT#404; END_IF;
(* Rung 83: Status Cycle Track202 *)
IF P_On AND Cyc_Track202.Step00 THEN DatAControl.OUT.CycleInformation := UINT#501; END_IF;
IF P_On AND Cyc_Track202.Step01 THEN DatAControl.OUT.CycleInformation := UINT#502; END_IF;
IF P_On AND Cyc_Track202.Step02 THEN DatAControl.OUT.CycleInformation := UINT#503; END_IF;
IF P_On AND Cyc_Track202.Step03 THEN DatAControl.OUT.CycleInformation := UINT#504; END_IF;
END_FUNCTION_BLOCK

FUNCTION_BLOCK FB_30052
VAR
    IS_TRack_201 : FB_101;
    I_Track201 : BOOL;  (* Input track 201 *)
    I_Track201DON : BOOL;  (* Input track 201 time delay on *)
    I_Track201DOFF : BOOL;  (* Input track 201 time delay off *)
    IS_Track_202 : FB_101;
    I_Track202 : BOOL;  (* input track 202 *)
    I_Track202DON : BOOL;  (* Input track 202 time delay on *)
    I_Track202DOFF : BOOL;  (* Input track 202 time delay off *)
    LS_Track_Up : FB_101;
    I_TrackUp : BOOL;  (* Input track up *)
    I_TrackUpDON : BOOL;  (* Input track up delay on *)
    LS_Track_Down : FB_101;
    I_TrackDown : BOOL;  (* Input track down *)
    I_TrackDownDON : BOOL;  (* Input track down delay on *)
    IS_Present : FB_101;
    I_Present : BOOL;  (* Input bench present *)
    I_PresentDON : BOOL;  (* Input present time delay on *)
    I_PresentDOFF : BOOL;  (* Input present delay off *)
    PB_Run_Motor : FB_101;
    I_PB_Run : BOOL;  (* Input pushbutton run motor *)
    MachineMode : ST_MachineMode;  (* Automatic Machine is automatic; SemiAutomatic Machine is semi automatic; Manual Machine is in manual *)
END_VAR
VAR RETAIN
    Cyc_Inb : ST_FB_30050_Cyc_Inbound;  (* Cycle inbound *)
    Cyc_Outb : ST_FB_30050_Cyc_Outbound;  (* Cycle outbound *)
    Cyc_Track_Inb : ST_FB_30052_Cyc_Track_Inbound;  (* Cycle track inbound *)
    Cyc_Track_Outb : ST_FB_30052_Cyc_Track_Outbound;  (* Cycle track outbound *)
END_VAR
VAR
    Instruction : FB_904;
    InstructionConditions : ST_Instruction_Conditions_Standaard;  (* Instruction conditions *)
    Start_Instruction : BOOL;  (* start instruction *)
    LoadGate : UINT;  (* Load gate *)
    UnloadGate : UINT;  (* unload gate *)
    Track_DirectionFromBuffer : BOOL;  (* Track direction from buffer *)
    Track_DirectionToBuffer : BOOL;  (* Track direction to buffer *)
    Reset_Alarm : BOOL;  (* Reset Alarm *)
    Reset_Cycle : BOOL;  (* Reset Cycle *)
    TransferOK : BOOL;  (* Transfer ok *)
    ConditionsFWD_OK : BOOL;  (* Conditions track forward ok *)
    ConditionsREV_OK : BOOL;  (* Conditions track reverse ok *)
    ConditionsGlobal_OK : BOOL;  (* Conditions global ok *)
    Track_Ref_FWD : BOOL;  (* Track reference is fwd *)
    Track_Ref_REV : BOOL;  (* Track reference is REV *)
    TrackMotor : FB_1011;
    M_Track_FWD : BOOL;  (* Motor track forward *)
    M_Track_REV : BOOL;  (* Motor track reverse *)
    Speed_Ref : INT;  (* Speed reference *)
    TrackUp_SA : BOOL;  (* Track up semi automatic *)
    Inverter_Track : FB_305;
    Beltmotor : FB_1011;
    Speed_Ref_Belt : INT;  (* Speed refeence belt *)
    Inverter_Belt : FB_305;
    M_Belt_FWD : BOOL;  (* Motor belt forward *)
    M_Belt_REV : BOOL;  (* Motor belt reverse *)
    Belt_Ref_Rev : BOOL;  (* Reference is reverse *)
    Belt_Ref_Fwd : BOOL;  (* Reference is forward *)
    ConditionsGlobal_Belt_Ok : BOOL;  (* Global conditions ok *)
    ConditionsFWD_Belt_Ok : BOOL;  (* Conditions forward ok *)
    COnditionsREV_Belt_Ok : BOOL;  (* Conditions reverse ok *)
    TrackInb_HighSpeedStart : BOOL;  (* Start timer high speed *)
    T_HighSpeed_TrackInb : _sTimer;  (* Timer highspeed *)
    TrackInb_Slow : BOOL;  (* track inbound slow *)
    TrackOutb_HighSpeedStart : BOOL;  (* Start timer high speed *)
    T_HighSpeed_TrackOutb : _sTimer;  (* Timer hig speed *)
    TrackOutbSlow : BOOL;  (* Track outbound slow *)
    Semi_Automatic_Track : FB_307;
    Track_SA_FWD : BOOL;  (* Track semi automatic forward *)
    Track_SA_REV : BOOL;  (* Track semi automatic reverse *)
    Semi_Automatic_Belt : FB_307;
    Belt_SA_FWD : BOOL;  (* Belt semi automatic forward *)
    Belt_SA_REV : BOOL;  (* Belt semi automatic reverse *)
    T_BeltSpeedHigh : _sTimer;  (* Timer belt hig speed *)
    MachineInAlarm : BOOL;  (* Machine has an alarm *)
    T_Warning_BridgeUp : _sTimer;
    T_Warning_BridgeDown : _sTimer;
    ResetTrack : BOOL;  (* Reset track *)
    T_NoGrantLeave : _sTimer;  (* Timer no grant leave *)
    T_NoContainer : _sTimer;  (* Timer no container *)
    V_Track_Ref : BOOL;  (* Track valve reference *)
    V_TrackV_Track_Ref : BOOL;
END_VAR
VAR_INPUT
    Enable : BOOL;
    EmergencyStopOk : BOOL;  (* Emergency stop OK *)
    MachineCode : UINT;  (* Machine code *)
    InverterStatus : ST_MX2\Status;  (* Inverterstatus *)
    Inputs : ST_FB_30050_Inputs;  (* IS_Track201 IS TRack 201; IS_Track202 IS track 202; IS_Present IS bench present; IS_PB_Run Pushbutton run motor *)
    Settings : ST_FB_30052_Settings;  (* TimeDelayON_IS201 Setting time delay on; TimeDelayOFF_IS201 Time delay off; TimeDelayON_IS202 Setting time delay on; TimeDelayOFF_IS202 Setting time delay off; TimeDelayON_LSTrackUp Setting time delay on; TimeDelayON_LSTrackDown Setting time delay on; TimeDelayON_ISPresent Setting time delay on; TimeDelayOFF_ISPresent Setting time delay off; TrackDirection Setting track direction 1 = to growroom, 2 = to workarea; MAX_Run_Time Max run time; MinSpeed Minimal speed; Inverter_NodeNumber_Track Node number track; Inverter_Parameters_Track Inverter parameters; MaxSpeed Max speed; TimeHighSpeed Setting timer; MaxSpeedBelt Max sped belt; TimeHighSpeedBelt Time high speed; DoTransferOutbound_101 Do transfer outbound *)
    CommIn101 : ST_FB_30051_CommInPipe;  (* SupplySignal Supply signal *)
    CommIn201 : ST_FB_30051_CommIn201;  (* SupplySignal Supply signal; RequestSignal Request signal *)
    CommIn202 : ST_FB_30051_CommIn202;  (* SupplySignal Supply signal; RequestSignal Request signal *)
END_VAR
VAR_OUTPUT
    OUT_InverterCommands : ST_MX2\Command;  (* Inverter commands *)
    OUT_InverterSpeed : INT;  (* Inverter speed *)
    Outputs : ST_FB_30052_Outputs;
    CommOut_101 : ST_FB_30051_CommOutPipe;  (* SupplySignal Supply signal; RequestSignal Request signal; SectionIsLow Section is low; StopOutbound Stop outbound *)
    CommOut_201 : ST_FB_30051_CommOut201;  (* SupplySignal Supply signal; RequestSignal request signal *)
    CommOut_202 : ST_FB_30051_CommOut202;  (* SupplySignal Supply signal; RequestSignal request signal *)
END_VAR
VAR_IN_OUT
    DatAControl : ST_DatAControl_Standard;  (* IN Dat A Control instruction; OUT.Instruction Dat A Control instruction out; OUT.Alarm04 Alarm word 4; IN.MachineMode Machine mode; IN.Settings.ResetAlarm Dat A Control Reset Alarm; IN.Settings.ResetCycle Dat A Control Reset Cycle; OUT.Alarm00 Alarm word 0; OUT.Alarm01 Alarm word 1; OUT.TotalDone Total done; OUT.Warning00 Warning word 0; OUT.Alarm02 Alarm word 2; OUT.CycleInformation Cycle information; OUT.Alarm03 Alarm word 3 *)
    Commands : ST_FB_30051_Commands;  (* Commands; BeltUp Commands belt up; BeltDown Commands belt down *)
    TransferBuffer : ST_TransferBuffer;  (* Transferbuffer *)
    Inverter_WriteParameters : BOOL;  (* Write parameters *)
    Inverter_WriteParametersDone : BOOL;  (* Write parameters done *)
END_VAR
VAR_EXTERNAL
    Dummy : BOOL;
    ES_OK : BOOL;
END_VAR
VAR
    _e1 : R_TRIG;
    _t2 : BOOL;
    _e3 : R_TRIG;
    _e4 : R_TRIG;
    _p5 : BOOL;
    _t6 : BOOL;
    _e7 : R_TRIG;
    _e8 : R_TRIG;
    _p9 : BOOL;
    _t10 : BOOL;
    _t11 : BOOL;
    _t12 : BOOL;
    _p13 : BOOL;
    _p14 : BOOL;
    _t15 : BOOL;
END_VAR
(* ladder, written here as Structured Text *)

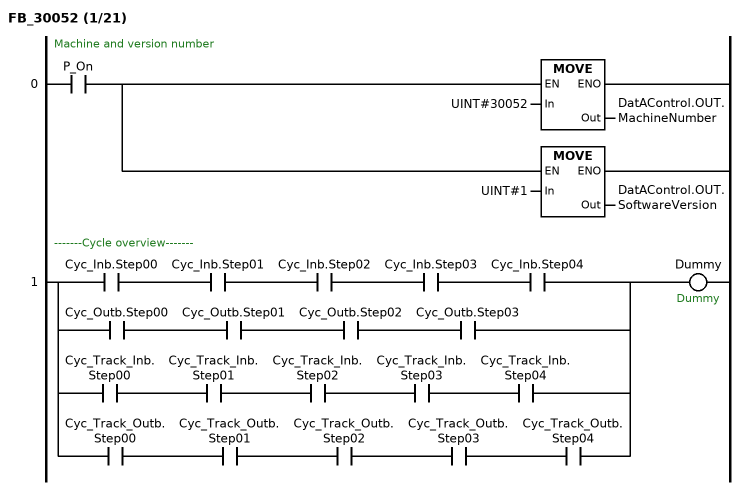
(* Rung 0: Machine and version number *)
IF P_On THEN
    DatAControl.OUT.MachineNumber := UINT#30052;
    DatAControl.OUT.SoftwareVersion := UINT#1;
END_IF;
(* Rung 1: -------Cycle overview------- *)
Dummy := (Cyc_Inb.Step00 AND Cyc_Inb.Step01 AND Cyc_Inb.Step02 AND Cyc_Inb.Step03 AND Cyc_Inb.Step04) OR (Cyc_Outb.Step00 AND Cyc_Outb.Step01 AND Cyc_Outb.Step02 AND Cyc_Outb.Step03) OR (Cyc_Track_Inb.Step00 AND Cyc_Track_Inb.Step01 AND Cyc_Track_Inb.Step02 AND Cyc_Track_Inb.Step03 AND Cyc_Track_Inb.Step04) OR (Cyc_Track_Outb.Step00 AND Cyc_Track_Outb.Step01 AND Cyc_Track_Outb.Step02 AND Cyc_Track_Outb.Step03 AND Cyc_Track_Outb.Step04);

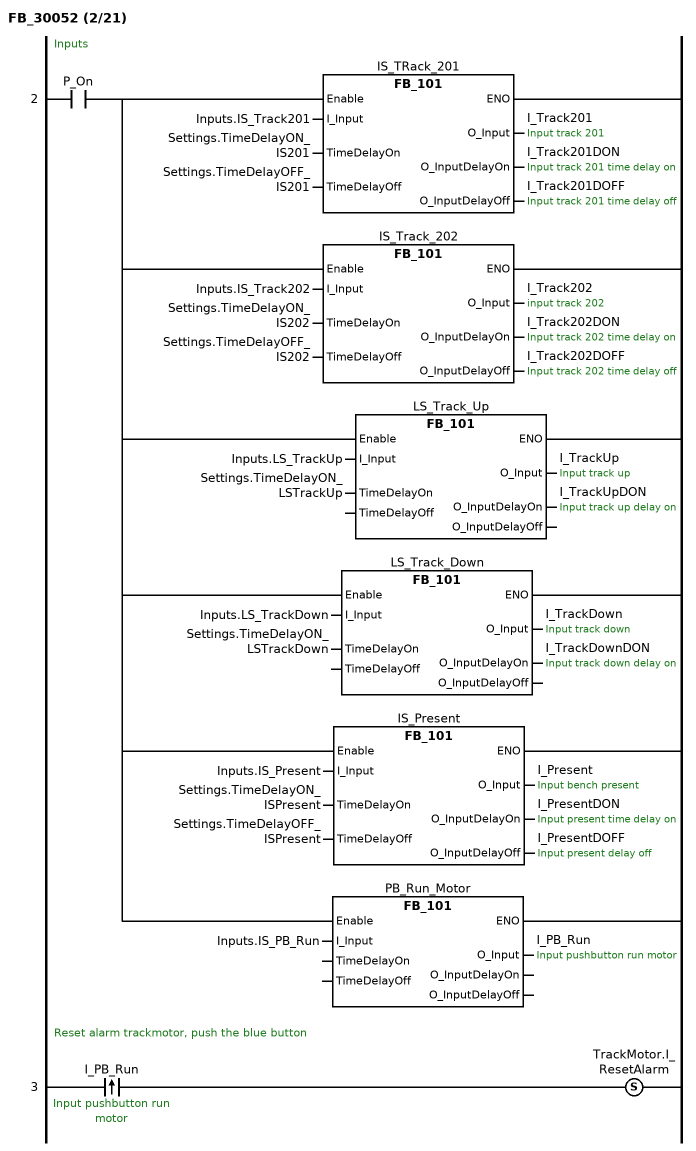
(* Rung 2: Inputs *)
IS_TRack_201(Enable := P_On, I_Input := Inputs.IS_Track201, TimeDelayOn := Settings.TimeDelayON_IS201, TimeDelayOff := Settings.TimeDelayOFF_IS201, O_Input => I_Track201, O_InputDelayOn => I_Track201DON, O_InputDelayOff => I_Track201DOFF);
IS_Track_202(Enable := P_On, I_Input := Inputs.IS_Track202, TimeDelayOn := Settings.TimeDelayON_IS202, TimeDelayOff := Settings.TimeDelayOFF_IS202, O_Input => I_Track202, O_InputDelayOn => I_Track202DON, O_InputDelayOff => I_Track202DOFF);
LS_Track_Up(Enable := P_On, I_Input := Inputs.LS_TrackUp, TimeDelayOn := Settings.TimeDelayON_LSTrackUp, O_Input => I_TrackUp, O_InputDelayOn => I_TrackUpDON);
LS_Track_Down(Enable := P_On, I_Input := Inputs.LS_TrackDown, TimeDelayOn := Settings.TimeDelayON_LSTrackDown, O_Input => I_TrackDown, O_InputDelayOn => I_TrackDownDON);
IS_Present(Enable := P_On, I_Input := Inputs.IS_Present, TimeDelayOn := Settings.TimeDelayON_ISPresent, TimeDelayOff := Settings.TimeDelayOFF_ISPresent, O_Input => I_Present, O_InputDelayOn => I_PresentDON, O_InputDelayOff => I_PresentDOFF);
PB_Run_Motor(Enable := P_On, I_Input := Inputs.IS_PB_Run, O_Input => I_PB_Run);
(* Rung 3: Reset alarm trackmotor, push the blue button *)
_e1(CLK := I_PB_Run);
IF _e1.Q THEN TrackMotor.I_ResetAlarm := TRUE; END_IF;

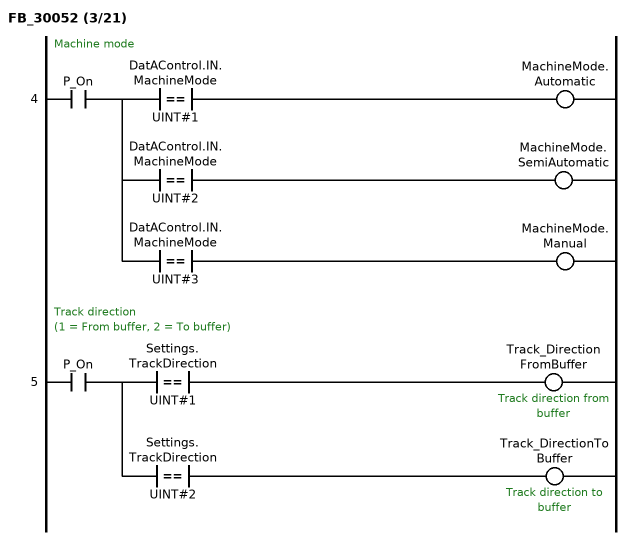
(* Rung 4: Machine mode *)
MachineMode.Automatic := P_On AND (DatAControl.IN.MachineMode = UINT#1);
MachineMode.SemiAutomatic := P_On AND (DatAControl.IN.MachineMode = UINT#2);
MachineMode.Manual := P_On AND (DatAControl.IN.MachineMode = UINT#3);
(* Rung 5: Track direction / (1 = From buffer, 2 = To buffer) *)
Track_DirectionFromBuffer := P_On AND (Settings.TrackDirection = UINT#1);
Track_DirectionToBuffer := P_On AND (Settings.TrackDirection = UINT#2);

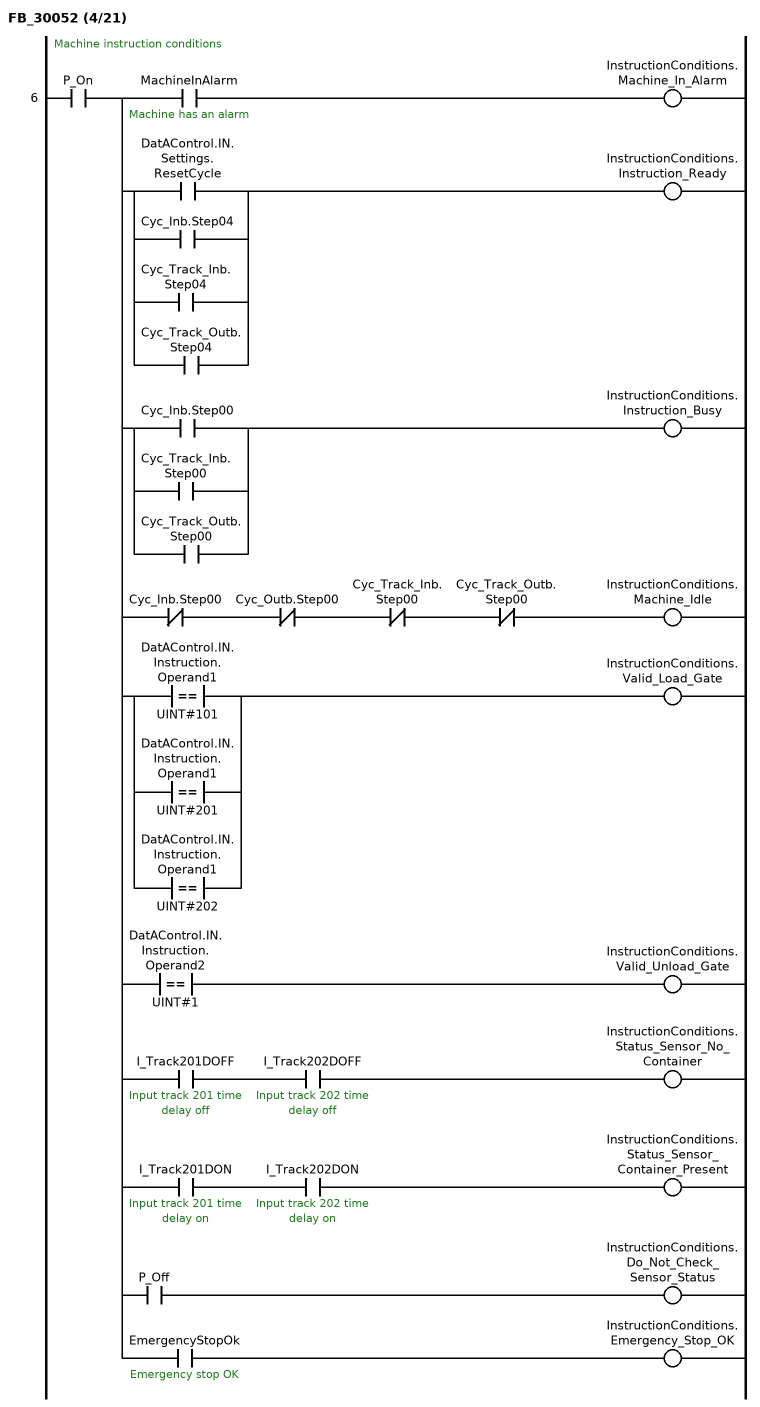
(* Rung 6: Machine instruction conditions *)
InstructionConditions.Machine_In_Alarm := P_On AND MachineInAlarm;
InstructionConditions.Instruction_Ready := P_On AND (DatAControl.IN.Settings.ResetCycle OR Cyc_Inb.Step04 OR Cyc_Track_Inb.Step04 OR Cyc_Track_Outb.Step04);
InstructionConditions.Instruction_Busy := P_On AND (Cyc_Inb.Step00 OR Cyc_Track_Inb.Step00 OR Cyc_Track_Outb.Step00);
InstructionConditions.Machine_Idle := P_On AND NOT Cyc_Inb.Step00 AND NOT Cyc_Outb.Step00 AND NOT Cyc_Track_Inb.Step00 AND NOT Cyc_Track_Outb.Step00;
InstructionConditions.Valid_Load_Gate := P_On AND ((DatAControl.IN.Instruction.Operand1 = UINT#101) OR (DatAControl.IN.Instruction.Operand1 = UINT#201) OR (DatAControl.IN.Instruction.Operand1 = UINT#202));
InstructionConditions.Valid_Unload_Gate := P_On AND (DatAControl.IN.Instruction.Operand2 = UINT#1);
InstructionConditions.Status_Sensor_No_Container := P_On AND I_Track201DOFF AND I_Track202DOFF;
InstructionConditions.Status_Sensor_Container_Present := P_On AND I_Track201DON AND I_Track202DON;
InstructionConditions.Do_Not_Check_Sensor_Status := P_On AND P_Off;
InstructionConditions.Emergency_Stop_OK := P_On AND EmergencyStopOk;

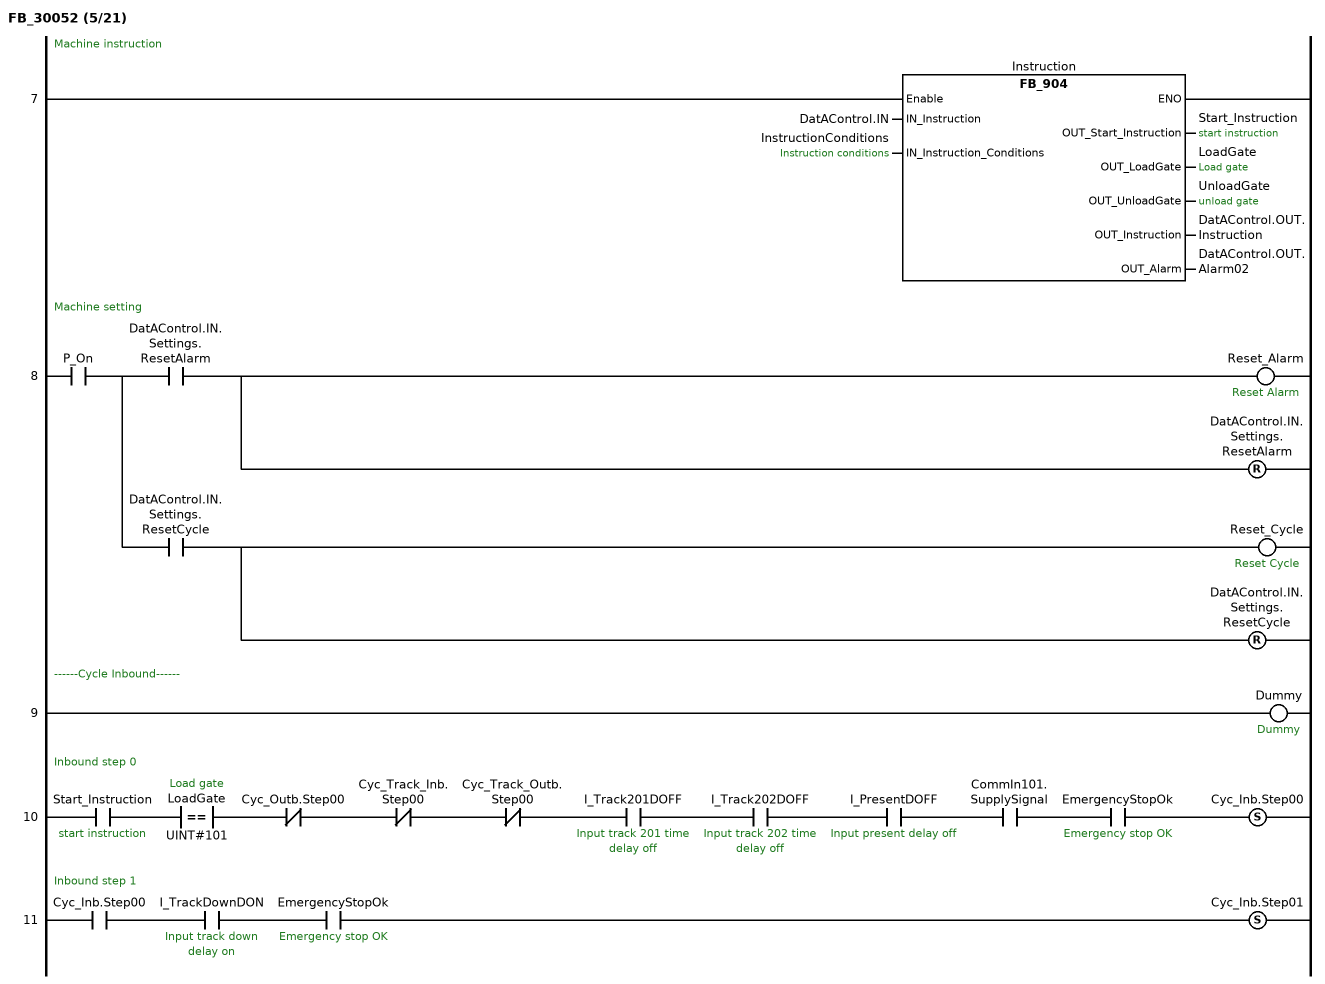
(* Rung 7: Machine instruction *)
Instruction(Enable := TRUE, IN_Instruction := DatAControl.IN, IN_Instruction_Conditions := InstructionConditions, OUT_Start_Instruction => Start_Instruction, OUT_LoadGate => LoadGate, OUT_UnloadGate => UnloadGate, OUT_Instruction => DatAControl.OUT.Instruction, OUT_Alarm => DatAControl.OUT.Alarm02);
(* Rung 8: Machine setting *)
Reset_Alarm := P_On AND DatAControl.IN.Settings.ResetAlarm;
IF P_On AND DatAControl.IN.Settings.ResetAlarm THEN DatAControl.IN.Settings.ResetAlarm := FALSE; END_IF;
Reset_Cycle := P_On AND DatAControl.IN.Settings.ResetCycle;
IF P_On AND DatAControl.IN.Settings.ResetCycle THEN DatAControl.IN.Settings.ResetCycle := FALSE; END_IF;
(* Rung 9: ------Cycle Inbound------ *)
Dummy := TRUE;
(* Rung 10: Inbound step 0 *)
IF Start_Instruction AND (LoadGate = UINT#101) AND NOT Cyc_Outb.Step00 AND NOT Cyc_Track_Inb.Step00 AND NOT Cyc_Track_Outb.Step00 AND I_Track201DOFF AND I_Track202DOFF AND I_PresentDOFF AND CommIn101.SupplySignal AND EmergencyStopOk THEN
    Cyc_Inb.Step00 := TRUE;
END_IF;
(* Rung 11: Inbound step 1 *)
IF Cyc_Inb.Step00 AND I_TrackDownDON AND EmergencyStopOk THEN Cyc_Inb.Step01 := TRUE; END_IF;

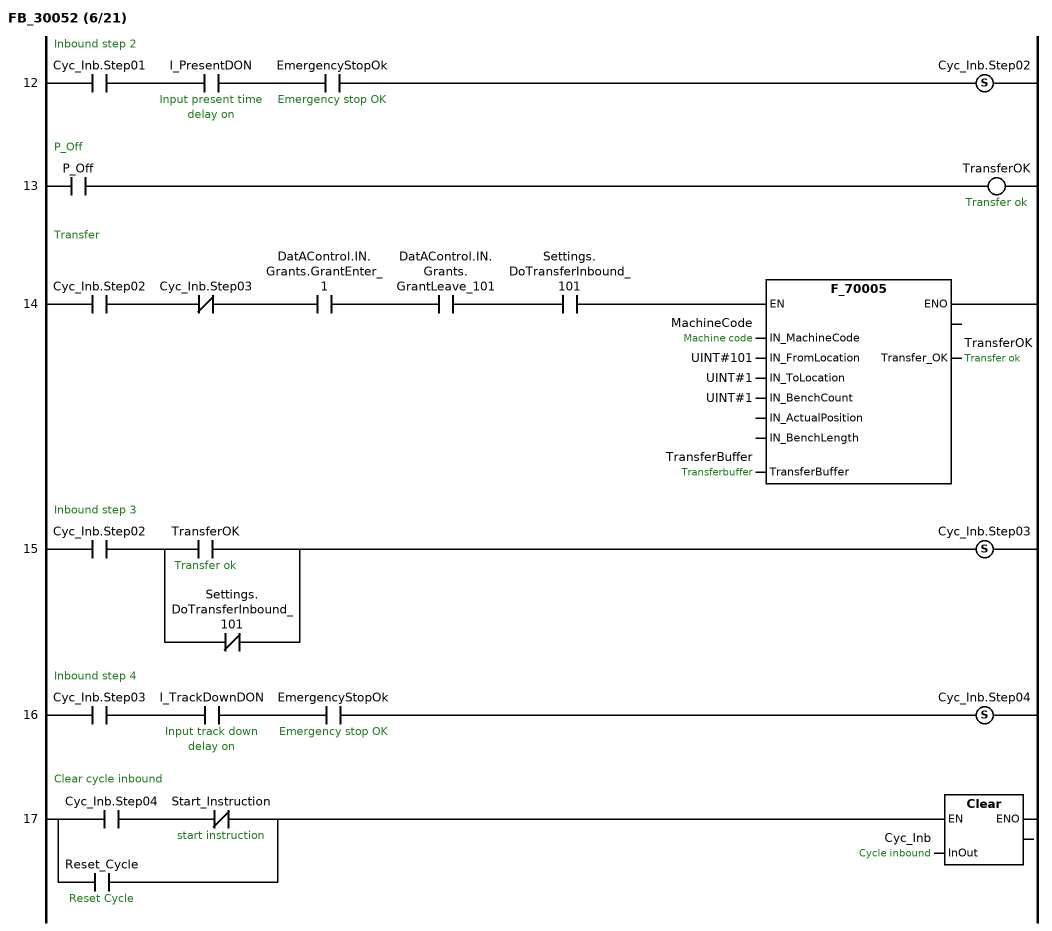
(* Rung 12: Inbound step 2 *)
IF Cyc_Inb.Step01 AND I_PresentDON AND EmergencyStopOk THEN Cyc_Inb.Step02 := TRUE; END_IF;
(* Rung 13: P_Off *)
TransferOK := P_Off;
(* Rung 14: Transfer *)
IF Cyc_Inb.Step02 AND NOT Cyc_Inb.Step03 AND DatAControl.IN.Grants.GrantEnter_1 AND DatAControl.IN.Grants.GrantLeave_101 AND Settings.DoTransferInbound_101 THEN
    F_70005(IN_MachineCode := MachineCode, IN_FromLocation := UINT#101, IN_ToLocation := UINT#1, IN_BenchCount := UINT#1, TransferBuffer := TransferBuffer, Transfer_OK => TransferOK);
END_IF;
(* Rung 15: Inbound step 3 *)
IF Cyc_Inb.Step02 AND (TransferOK OR NOT Settings.DoTransferInbound_101) THEN
    Cyc_Inb.Step03 := TRUE;
END_IF;
(* Rung 16: Inbound step 4 *)
IF Cyc_Inb.Step03 AND I_TrackDownDON AND EmergencyStopOk THEN Cyc_Inb.Step04 := TRUE; END_IF;
(* Rung 17: Clear cycle inbound *)
IF (Cyc_Inb.Step04 AND NOT Start_Instruction) OR Reset_Cycle THEN Clear(InOut := Cyc_Inb); END_IF;

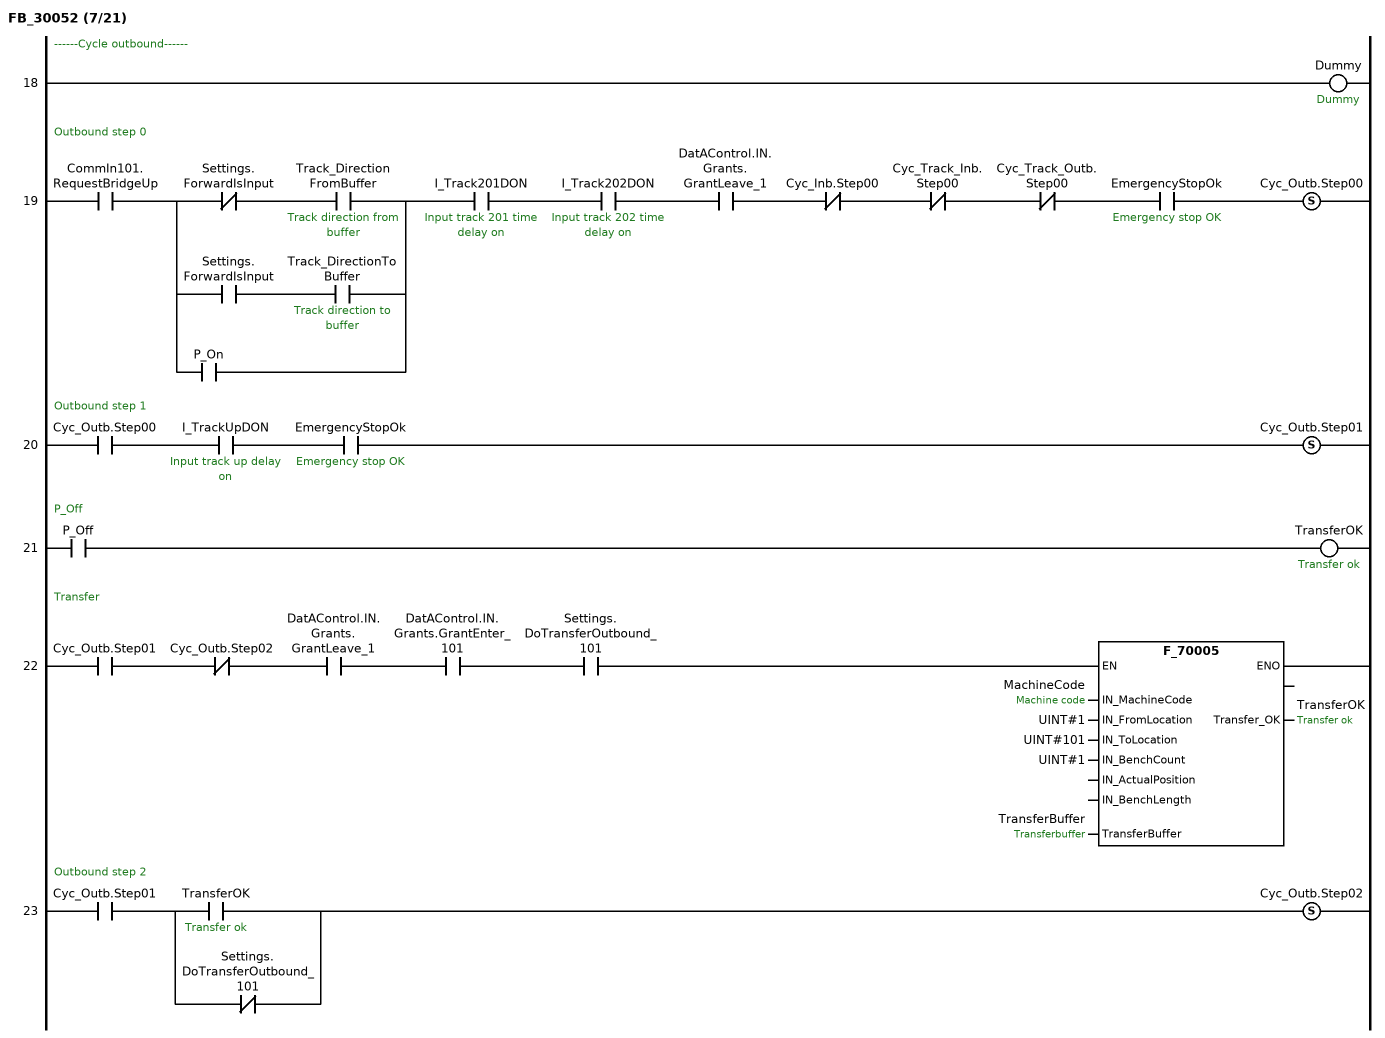
(* Rung 18: ------Cycle outbound------ *)
Dummy := TRUE;
(* Rung 19: Outbound step 0 *)
IF CommIn101.RequestBridgeUp AND ((NOT Settings.ForwardIsInput AND Track_DirectionFromBuffer) OR (Settings.ForwardIsInput AND Track_DirectionToBuffer) OR P_On) AND I_Track201DON AND I_Track202DON AND DatAControl.IN.Grants.GrantLeave_1 AND NOT Cyc_Inb.Step00 AND NOT Cyc_Track_Inb.Step00 AND NOT Cyc_Track_Outb.Step00 AND EmergencyStopOk THEN
    Cyc_Outb.Step00 := TRUE;
END_IF;
(* Rung 20: Outbound step 1 *)
IF Cyc_Outb.Step00 AND I_TrackUpDON AND EmergencyStopOk THEN Cyc_Outb.Step01 := TRUE; END_IF;
(* Rung 21: P_Off *)
TransferOK := P_Off;
(* Rung 22: Transfer *)
IF Cyc_Outb.Step01 AND NOT Cyc_Outb.Step02 AND DatAControl.IN.Grants.GrantLeave_1 AND DatAControl.IN.Grants.GrantEnter_101 AND Settings.DoTransferOutbound_101 THEN
    F_70005(IN_MachineCode := MachineCode, IN_FromLocation := UINT#1, IN_ToLocation := UINT#101, IN_BenchCount := UINT#1, TransferBuffer := TransferBuffer, Transfer_OK => TransferOK);
END_IF;
(* Rung 23: Outbound step 2 *)
IF Cyc_Outb.Step01 AND (TransferOK OR NOT Settings.DoTransferOutbound_101) THEN
    Cyc_Outb.Step02 := TRUE;
END_IF;

